// TIA Portal V19 program export: 9 tag tables, 2 data types, 63 data blocks, 26 code blocks (in call order from the OBs), 0 instance data blocks

VAR_GLOBAL   // PLC tag table "Default tag table"
   "System_Byte(1)" AT %MB1 : Byte;
   "Clock_Byte(1)" AT %MB0 : Byte;
   "Clock_10Hz(1)" AT %M0.0 : Bool;
   "Clock_5Hz(1)" AT %M0.1 : Bool;
   "Clock_2.5Hz(1)" AT %M0.2 : Bool;
   "Clock_2Hz(1)" AT %M0.3 : Bool;
   "Clock_1.25Hz(1)" AT %M0.4 : Bool;
   "Clock_1Hz(1)" AT %M0.5 : Bool;
   "Clock_0.625Hz(1)" AT %M0.6 : Bool;
   "Clock_0.5Hz(1)" AT %M0.7 : Bool;
END_VAR

VAR_GLOBAL   // PLC tag table "TT - Clocks"
   Clock_Byte AT %MB255 : Byte;
   Clock_10Hz AT %M255.0 : Bool;
   Clock_5Hz AT %M255.1 : Bool;
   "Clock_2.5Hz" AT %M255.2 : Bool;
   Clock_2Hz AT %M255.3 : Bool;
   "Clock_1.25Hz" AT %M255.4 : Bool;
   Clock_1Hz AT %M255.5 : Bool;
   "Clock_0.625Hz" AT %M255.6 : Bool;
   "Clock_0.5Hz" AT %M255.7 : Bool;
END_VAR

VAR_GLOBAL   // PLC tag table "TT - System"
   System_Byte AT %MB254 : Byte;
   FirstScan AT %M254.0 : Bool;
   DiagStatusUpdate AT %M254.1 : Bool;
   AlwaysTRUE AT %M254.2 : Bool;
   AlwaysFALSE AT %M254.3 : Bool;
END_VAR

VAR_GLOBAL   // PLC tag table "TT - Feeding"
   iFeedingSenCilOut_k1 AT %I2.4 : Bool;
   iFeedingSenLoaded AT %I2.5 : Bool;
   "oFeedingVenCilOut_K+" AT %Q1.5 : Bool;
END_VAR

VAR_GLOBAL   // PLC tag table "TT - General"
   iDkStart_S2 AT %I0.0 : Bool;   // NO
   iDkStop_S3 AT %I0.1 : Bool;   // NC
   iSelSchMan_Q2 AT %I0.2 : Bool;
   iDkReset_S4 AT %I0.3 : Bool;   // NO (reset VR)
   iStsNoodstop_S1 AT %I2.7 : Bool;   // NO
   oLmpAlarm_H1 AT %Q0.0 : Bool;
   oLmpWarningLowMaterial_H2 AT %Q1.7 : Bool;
   iSenPressure AT %I2.6 : Bool;   // true when pressure
END_VAR

VAR_GLOBAL   // PLC tag table "TT - Loading"
   iLoadingSenDown_a1 AT %I0.4 : Bool;
   iLoadingSenUp_a0 AT %I0.5 : Bool;
   iLoadingSenAtPick_b0 AT %I0.6 : Bool;
   iLoadingSenAtPlace_b1 AT %I0.7 : Bool;
   "oLoadingVenCilDown_A+" AT %Q0.1 : Bool;
   oLoadingVenCilPlace_B AT %Q0.2 : Bool;
   oLoadingVenGrip_C AT %Q0.3 : Bool;
END_VAR

VAR_GLOBAL   // PLC tag table "TT - Plate"
   iPlateSenCilPushingIn_d0 AT %I1.0 : Bool;   // Terugkoppeling pusher roteren plaat
   iPlateSenInductive_dm AT %I1.6 : Bool;   // True when metallic
   iPlateSenPresence_dp AT %I1.7 : Bool;
   iPlateSenNotBlack AT %I2.0 : Bool;   // Niet definitief, True when nothing and white
   "oPlateVenCilPushing_D+" AT %Q0.4 : Bool;
   "oPlateVenCilLocking_E+" AT %Q0.5 : Bool;
   "oPlateVenCilMeasuringDown_L+" AT %Q1.6 : Bool;
   iPlateSenHeight AT %IW65 : Int;
END_VAR

VAR_GLOBAL   // PLC tag table "TT - Reject"
   iRejectSenCilIn_f0 AT %I1.1 : Bool;
   iRejectSenCilOut_f1 AT %I1.2 : Bool;
   iRejectSenCilUp_g0 AT %I1.3 : Bool;
   "oRejectVenCilOut_F+" AT %Q0.6 : Bool;   // Bistabiel
   "oRejectVenCilIn_F-" AT %Q0.7 : Bool;   // Bistabiel
   oRejectVenCilDown_E AT %Q1.0 : Bool;
   "oRejectVenVacuum_V+" AT %Q1.1 : Bool;
   "iRejectSenVacuum_V+" AT %I2.1 : Bool;   // true when vacuum
END_VAR

VAR_GLOBAL   // PLC tag table "TT - Transport"
   iTransportSenDown_h1 AT %I1.4 : Bool;
   iTransportSenUp_h0 AT %I1.5 : Bool;
   iTransportSenAtPlate_i0 AT %I2.2 : Bool;
   iTransportSenAtCart_i1 AT %I2.3 : Bool;
   "oTransportVenCilDown_A+" AT %Q1.2 : Bool;
   "oTransportVenCilCart_I+" AT %Q1.3 : Bool;
   "oTransportVenGripClosed_J+" AT %Q1.4 : Bool;
END_VAR

TYPE "UDT_Recipe"
VERSION : 0.1
   STRUCT
      "Type" : Int;
      Aantal : Int;
      Progress : Int;
   END_STRUCT;

END_TYPE

TYPE "UDT_coverProperties"
VERSION : 0.1
   STRUCT
      loaded : Bool;   // Indicates that there is an item in the current location
      reject : Bool;   // Indicates that the current item is to be rejected
      properties : Struct
         metallic : Bool;   // Indicates that the current item is metallic
         notBlack : Bool;   // Indicates that the current item is not black
         correctOrientation : Bool;   // Indicates that the current item has the correct orientation
      END_STRUCT;
   END_STRUCT;

END_TYPE

DATA_BLOCK "DB_Alarm"
{ S7_Optimized_Access := 'TRUE' }
VERSION : 0.1
NON_RETAIN
   VAR 
      com : Struct   // Alarms from Transfer PLC communication
         S7_PUTerr : Bool;   // Error reported by PUT instruction
         S7_GETerr : Bool;   // Error reported by GET instruction
         WD : Bool;   // Watchdog timed out
      END_STRUCT;
      general : Struct   // General alarms
         global : Bool;   // Indicates that an alarm is active
         emergencyStop : Bool;   // Indicates that the emergency stop button is activated
         airPressure : Bool;   // Indicates a loss in air pressure
      END_STRUCT;
      feeding : Struct   // Alarms generated by the "Feeding" EM
         materialLow : Bool;   // Indicates an empty mag
      END_STRUCT;
      reject : Struct   // Alarms generated by the "Reject" EM
         vacuum : Bool;   // Indicates loss of vacuum when not expected
      END_STRUCT;
   END_VAR


BEGIN

END_DATA_BLOCK

DATA_BLOCK "DB_Global"
{ S7_Optimized_Access := 'TRUE' }
VERSION : 0.1
NON_RETAIN
   VAR 
      com : Struct   // Communication state object
         WD : Int;   // Watchdog mem for S7 communication with Transfer PLC
      END_STRUCT;
      general : Struct   // General state object
         startup : Bool;   // Indicates "startup" mode
         started : Bool;   // Indicates "started" mode
         man : Bool;   // Indicates "manual" mode
         resetSignal : Bool;   // Gives the reset signal (1s high)
         init : Bool;   // Sets the "Global Grafcet" to step 0
         DEBUG_AlwaysFalse : Bool;   // Used for debugging
         DEBUG_AlwaysTrue : Bool;   // Used for debugging
      END_STRUCT;
      feeding : Struct   // Feeding state object
         init : Bool;   // Sets the "Feeding Grafcet" to step 0
         sigReadyToReload : Bool;   // Indicates that "Feeding Grafcet" is ready
      END_STRUCT;
      loading : Struct   // Loading state object
         init : Bool;   // Sets the "Loading Grafcet" to step 0
         cmdPlaceNewCover : Bool;   // Command to start the "Loading" process
         sigReadyToPlace : Bool;   // Indicates that "Loading Grafcet" is ready
      END_STRUCT;
      plate : Struct   // Loading state object
         currentCovers { S7_SetPoint := 'False'} : Array[0..7] of "UDT_coverProperties";   // Array with all the data for the locations on the plate
         init_rotate : Bool;   // Sets the "Rotate Grafcet" to step 0
         cmdRotate : Bool;   // Command to start the "Rotate" process
         sigReadyToRotate : Bool;   // Indicates that "Rotate Grafcet" is ready
         init_measure : Bool;   // Sets the "Measure Grafcet" to step 0
         cmdMeasure : Bool;   // Command to start the "Measure" process
         sigReadyToMeasure : Bool;   // Indicates that "Measure Grafcet" is ready
      END_STRUCT;
      reject : Struct   // Reject state object
         init : Bool;   // Sets the "Reject Grafcet" to step 0
         cmdReject : Bool;   // Command to start the "Reject" process
         sigReadyToReject : Bool;   // Indicates that "Reject Grafcet" is ready
      END_STRUCT;
      transport : Struct   // Transport state object
         init : Bool;   // Sets the "Transport Grafcet" to step 0
         cmdTransport : Bool;   // Command to start the "Transport" process
         sigReadyToTransport : Bool;   // Indicates that "Transport Grafcet" is ready
      END_STRUCT;
   END_VAR


BEGIN

END_DATA_BLOCK

DATA_BLOCK "DB_IO"
{ S7_Optimized_Access := 'TRUE' }
VERSION : 0.1
NON_RETAIN
   VAR 
      general : Struct   // IO dedicated to no specific EM
         iDkStart : Bool;   // Processed input value
         iDkStop : Bool;   // Processed input value
         iSelSchMan : Bool;   // Processed input value
         iDkReset : Bool;   // Processed input value
         iSenPressure : Bool;   // Processed input value
         iStsNoodstop : Bool;   // Processed input value
         oLmpAlarm : Bool;   // Automatic output value
         oLmpWarningLowMaterial : Bool;   // Automatic output value
      END_STRUCT;
      feeding : Struct   // IO dedicated to Feeding EM
         iFeedingSenCilOut_k1 : Bool;   // Processed input value
         iFeedingSenLoaded : Bool;   // Processed input value
         "oFeedingVenCilOut_K+" : Bool;   // Automatic output value
      END_STRUCT;
      loading : Struct   // IO dedicated to Loading EM
         iLoadingSenDown : Bool;   // Processed input value
         iLoadingSenUp : Bool;   // Processed input value
         iLoadingSenAtPick : Bool;   // Processed input value
         iLoadingSenAtPlace : Bool;   // Processed input value
         oLoadingVenCilDown : Bool;   // Automatic output value
         oLoadingVenCilPlace : Bool;   // Automatic output value
         oLoadingVenGrip : Bool;   // Automatic output value
      END_STRUCT;
      plate : Struct   // IO dedicated to Plate EM
         iPlateSenCilPushingIn : Bool;   // Processed input value
         iPlateSenInductive : Bool;   // Processed input value
         iPlateSenPresence : Bool;   // Processed input value
         iPlateSenNotBlack : Bool;   // Processed input value
         iPlateSenHeight : Int;   // Processed input value
         oPlateVenCilPushing : Bool;   // Automatic output value
         oPlateVenCilLocking : Bool;   // Automatic output value
         oPlateVenCilMeasuringDown : Bool;   // Automatic output value
      END_STRUCT;
      reject : Struct   // IO dedicated to Reject EM
         iRejectSenCilIn : Bool;   // Processed input value
         iRejectSenCilOut : Bool;   // Processed input value
         iRejectSenCilUp : Bool;   // Processed input value
         iRejectSenVacuum : Bool;   // Processed input value
         oRejectVenCilOut : Bool;   // Automatic output value
         oRejectVenCilIn : Bool;   // Automatic output value
         oRejectVenCilDown : Bool;   // Automatic output value
         oRejectVenVacuum : Bool;   // Automatic output value
      END_STRUCT;
      transport : Struct   // IO dedicated to Transport EM
         iTransportSenDown : Bool;   // Processed input value
         iTransportSenUp : Bool;   // Processed input value
         iTransportSenAtPlate : Bool;   // Processed input value
         iTransportSenAtCart : Bool;   // Processed input value
         oTransportVenCilDown : Bool;   // Automatic output value
         oTransportVenCilCart : Bool;   // Automatic output value
         oTransportVenGripClosed : Bool;   // Automatic output value
      END_STRUCT;
   END_VAR


BEGIN

END_DATA_BLOCK

DATA_BLOCK "DB_Testing"
{ S7_Optimized_Access := 'TRUE' }
VERSION : 0.1
NON_RETAIN
   VAR 
      enable : Struct
         TransferPLC : Bool;   // Enables or disables the entire FB for testing purposes only
         GlobalGrafcet : Bool;   // Enables or disables the entire FB for testing purposes only
         Feeding : Bool;   // Enables or disables the entire FB for testing purposes only
         Loading : Bool;   // Enables or disables the entire FB for testing purposes only
         Rotate : Bool;   // Enables or disables the entire FB for testing purposes only
         Measure : Bool;   // Enables or disables the entire FB for testing purposes only
         Reject : Bool;   // Enables or disables the entire FB for testing purposes only
         Transport : Bool;   // Enables or disables the entire FB for testing purposes only
      END_STRUCT;
      init : Struct
         GlobalGrafcet : Bool;   // Sets current step to 0 (rising edge)
         Feeding : Bool;   // Sets current step to 0 (rising edge)
         Loading : Bool;   // Sets current step to 0 (rising edge)
         Rotate : Bool;   // Sets current step to 0 (rising edge)
         Measure : Bool;   // Sets current step to 0 (rising edge)
         Reject : Bool;   // Sets current step to 0 (rising edge)
         Transport : Bool;   // Sets current step to 0 (rising edge)
      END_STRUCT;
      value : Struct
         RecipeType : Int;   // Emulates current recipe to be 1 or 2 for testing purposes only
         RejectBit : Bool;   // Emulates that the current cover needs to be rejected
         CoverLoaded : Bool;   // Emulates that the location is loaded
      END_STRUCT;
      signal : Struct
         Transfer_CarrierReady : Bool;   // Emulates "carrierReady" signal from transfer PLC for testing purposes only
         Feeding_ReadyToReload : Bool;
         Loading_ReadyToPlace : Bool;
         Plate_ReadyToRotate : Bool;
         Plate_ReadyToMeasure : Bool;
         Reject_ReadyToReject : Bool;
         Transport_ReadyToTransport : Bool;
      END_STRUCT;
      cmd : Struct
         Loading : Bool;
         Plate_Rotate : Bool;
         Plate_Measure : Bool;
         Reject : Bool;
         Transport : Bool;
      END_STRUCT;
   END_VAR


BEGIN
   enable.TransferPLC := false;
   enable.GlobalGrafcet := false;
   enable.Feeding := false;
   enable.Loading := false;
   enable.Rotate := false;
   enable.Measure := false;
   enable.Reject := false;
   enable.Transport := false;
   init.GlobalGrafcet := false;
   init.Feeding := false;
   init.Loading := false;
   init.Rotate := false;
   init.Measure := false;
   init.Reject := false;
   init.Transport := false;
   value.RecipeType := 0;
   value.RejectBit := false;
   value.CoverLoaded := false;
   signal.Transfer_CarrierReady := false;
   signal.Feeding_ReadyToReload := false;
   signal.Loading_ReadyToPlace := false;
   signal.Plate_ReadyToRotate := false;
   signal.Plate_ReadyToMeasure := false;
   signal.Reject_ReadyToReject := false;
   signal.Transport_ReadyToTransport := false;
   cmd.Loading := false;
   cmd.Plate_Rotate := false;
   cmd.Plate_Measure := false;
   cmd.Reject := false;
   cmd.Transport := false;

END_DATA_BLOCK

DATA_BLOCK "DB_MES"
{ S7_Optimized_Access := 'FALSE' }
VERSION : 0.1
NON_RETAIN
   STRUCT 
      "IO van FB_ControlRecipes" : Struct
         iNewRecipe : Bool;
         iNewType : Int;
         iNewAantal : Int;
         iRemoveRecipe : Bool;
         iRecipeToBeRemoved : Int;
         iReceptKlaar : Bool;
         oFull : Bool;
         oEmpty : Bool;
      END_STRUCT;
      Algemeen : Struct
         mReceptGestart : Bool;
         mReceptActief : Bool;
         mInstallatieGestart : Bool;
         mWatchdogPLC : Int;
         mAlmActive : Bool;
      END_STRUCT;
      Alarmen : Struct
         mAlmGlobal : Bool;
         mAlmEmergencyStop : Bool;
         mAlmAirPressureLow : Bool;
         mAlmMaterialLow : Bool;
         mAlmVacuum : Bool;
      END_STRUCT;
      Merkers : Struct
         mMerkerSR1 : Bool;
         mMerkerSR2 : Bool;
      END_STRUCT;
   END_STRUCT;


BEGIN

END_DATA_BLOCK

DATA_BLOCK "DB_Recipes"
{ S7_Optimized_Access := 'FALSE' }
VERSION : 0.1
NON_RETAIN
   STRUCT 
      Recipes { S7_SetPoint := 'False'} : Array[0..4] of "UDT_Recipe";
   END_STRUCT;


BEGIN

END_DATA_BLOCK

DATA_BLOCK "FB_ControlRecipes_DB"
{ S7_Optimized_Access := 'TRUE' }
VERSION : 0.1
NON_RETAIN
"FB_ControlRecipes"

BEGIN

END_DATA_BLOCK

DATA_BLOCK "DB_HMI"
{ S7_Optimized_Access := 'TRUE' }
VERSION : 0.1
NON_RETAIN
   VAR 
      general : Struct
         read_fromPLC : Struct
            Gestart : Bool;
            Gestopt : Bool;
            Storing : Bool;
            Man : Bool;
            Auto : Bool;
         END_STRUCT;
         alarmen : Struct
            Emergency : Bool;
            AirPressure : Bool;
         END_STRUCT;
         write_toPLC : Struct
            Cmd_Start : Bool;   // Om te sturen in Auto
            Cmd_Stop : Bool;   // Om te sturen in Auto
            Cmd_Reset : Bool;   // Om te sturen in Auto
            Cmd_Init : Bool;
         END_STRUCT;
      END_STRUCT;
      feeding : Struct
         read_fromPLC : Struct
            SenLoaded : Bool;
            SenCilOut_k1 : Bool;
            MagazijnLeeg : Bool;
         END_STRUCT;
         alarmen : Struct
            MaterialLow : Bool;
         END_STRUCT;
         write_toPLC : Struct
            Man_Out : Bool;
         END_STRUCT;
      END_STRUCT;
      loading : Struct
         read_fromPLC : Struct
            SenDown_a1 : Bool;
            SenUp_a0 : Bool;
            SenAtPick_b0 : Bool;
            SenAtPlace_b1 : Bool;
            oGrip : Bool;   // Inlezen om weer te geven wat deze doet
         END_STRUCT;
         alarmen : Struct
            CilDownTimeout : Bool;
            CilPlaceTimeout : Bool;
         END_STRUCT;
         write_toPLC : Struct
            Man_Grip : Bool;
            Man_Down : Bool;
            Man_Place : Bool;
         END_STRUCT;
      END_STRUCT;
      plate : Struct
         read_fromPLC : Struct
            oLock : Bool;   // Inlezen om weer te geven wat deze doet
            SenCilPushIn : Bool;   // cylinder terug (not pushed) true
            oMeasureDown : Bool;   // cylinder uit Measure
            MeasureDownNOK : Bool;   // Berekend
            MeasureDownOK : Bool;   // Berekend
         END_STRUCT;
         alarmen : Struct
            CilMeasureTime : Bool;
         END_STRUCT;
         write_toPLC : Struct
            Man_Measure : Bool;
            Man_Push : Bool;
            Man_Lock : Bool;
         END_STRUCT;
      END_STRUCT;
      reject : Struct
         read_fromPLC : Struct
            SenVacuüm : Bool;
            SenOut : Bool;
            SenIn : Bool;
            SenUp : Bool;
         END_STRUCT;
         alarmen : Struct
            CilOutTime : Bool;
            Vacuüm : Bool;
         END_STRUCT;
         write_toPLC : Struct
            Man_Out : Bool;
            Man_Vacuüm : Bool;
            Man_Down : Bool;
         END_STRUCT;
      END_STRUCT;
      transport : Struct
         read_fromPLC : Struct
            oGrip : Bool;   // inlezen om weer te geven wat deze doet
            CilUp : Bool;
            CilDown : Bool;
            CilPick : Bool;
            CilPlace : Bool;
         END_STRUCT;
         alarmen : Struct
            CilDownTime : Bool;
            CilPlaceTime : Bool;
         END_STRUCT;
         write_toPLC : Struct
            Man_Grip : Bool;
            Man_Down : Bool;
            Man_Place : Bool;
         END_STRUCT;
      END_STRUCT;
   END_VAR


BEGIN

END_DATA_BLOCK

DATA_BLOCK "DB_TransferPLC"
{ S7_Optimized_Access := 'TRUE' }
VERSION : 0.1
NON_RETAIN
   VAR 
      Watchdog : Int;   // value between 0 and 20000 that counts up every second
      CarrierReady : Bool;   // inidcates if the carrier is in place and ready to recieve a cover
      ItemPlaced : Bool;   // indicates if the cover station has placed the cover on the carrier
   END_VAR


BEGIN

END_DATA_BLOCK

DATA_BLOCK "ID_PE_GlobalGrafcet"
{ S7_Optimized_Access := 'TRUE' }
VERSION : 0.1
NON_RETAIN
"FB_PE_GlobalGrafcet"

BEGIN

END_DATA_BLOCK

DATA_BLOCK "ID_PE_Feeding_Grafcet"
{ S7_Optimized_Access := 'TRUE' }
VERSION : 0.1
NON_RETAIN
"FB_PE_Feeding_Grafcet"

BEGIN

END_DATA_BLOCK

DATA_BLOCK "ID_PE_Loading_Grafcet"
{ S7_Optimized_Access := 'TRUE' }
VERSION : 0.1
NON_RETAIN
"FB_PE_Loading"

BEGIN

END_DATA_BLOCK

DATA_BLOCK "ID_PE_Plate_Grafcet"
{ S7_Optimized_Access := 'TRUE' }
VERSION : 0.1
NON_RETAIN
"FB_PE_Plate_Rotate"

BEGIN

END_DATA_BLOCK

DATA_BLOCK "ID_PE_Plate_Measure"
{ S7_Optimized_Access := 'TRUE' }
VERSION : 0.1
NON_RETAIN
"FB_PE_Plate_Measure"

BEGIN

END_DATA_BLOCK

DATA_BLOCK "ID_PE_Reject"
{ S7_Optimized_Access := 'TRUE' }
VERSION : 0.1
NON_RETAIN
"FB_PE_Reject"

BEGIN

END_DATA_BLOCK

DATA_BLOCK "ID_PE_Transport"
{ S7_Optimized_Access := 'TRUE' }
VERSION : 0.1
NON_RETAIN
"FB_PE_Transport"

BEGIN

END_DATA_BLOCK

DATA_BLOCK "ID_Algemeen_CM_DI_iDkReset"
{ S7_Optimized_Access := 'FALSE' }
VERSION : 0.1
NON_RETAIN
"FB_CM_DI_Sensor"

BEGIN

END_DATA_BLOCK

DATA_BLOCK "ID_Algemeen_CM_DI_iDkStart"
{ S7_Optimized_Access := 'FALSE' }
VERSION : 0.1
NON_RETAIN
"FB_CM_DI_Sensor"

BEGIN

END_DATA_BLOCK

DATA_BLOCK "ID_Algemeen_CM_DI_iDkStop"
{ S7_Optimized_Access := 'FALSE' }
VERSION : 0.1
NON_RETAIN
"FB_CM_DI_Sensor"

BEGIN

END_DATA_BLOCK

DATA_BLOCK "ID_Algemeen_CM_DI_iSelSchMan"
{ S7_Optimized_Access := 'FALSE' }
VERSION : 0.1
NON_RETAIN
"FB_CM_DI_Sensor"

BEGIN

END_DATA_BLOCK

DATA_BLOCK "ID_Algemeen_CM_DI_iStsNoodstop"
{ S7_Optimized_Access := 'FALSE' }
VERSION : 0.1
NON_RETAIN
"FB_CM_DI_Sensor"

BEGIN

END_DATA_BLOCK

DATA_BLOCK "ID_Algemeen_PE_StartStop"
{ S7_Optimized_Access := 'FALSE' }
VERSION : 0.1
NON_RETAIN
"FB_PE_StartStop"

BEGIN

END_DATA_BLOCK

DATA_BLOCK "ID_CM_Lamp_Alarm_H1"
{ S7_Optimized_Access := 'TRUE' }
VERSION : 0.1
NON_RETAIN
"FB_CM_Lamp_1200"

BEGIN

END_DATA_BLOCK

DATA_BLOCK "ID_Feeding_CM_DI_SenCilOut"
{ S7_Optimized_Access := 'FALSE' }
VERSION : 0.1
NON_RETAIN
"FB_CM_DI_Sensor"

BEGIN

END_DATA_BLOCK

DATA_BLOCK "ID_Feeding_CM_DI_SenLoaded"
{ S7_Optimized_Access := 'FALSE' }
VERSION : 0.1
NON_RETAIN
"FB_CM_DI_Sensor"

BEGIN

END_DATA_BLOCK

DATA_BLOCK "ID_Feeding_CM_oFeedingVenCilOut"
{ S7_Optimized_Access := 'FALSE' }
VERSION : 0.1
NON_RETAIN
"FB_CM_Cilinder"

BEGIN

END_DATA_BLOCK

DATA_BLOCK "ID_Loading_CM_DI_iLoadingSenAtPick_b0"
{ S7_Optimized_Access := 'FALSE' }
VERSION : 0.1
NON_RETAIN
"FB_CM_DI_Sensor"

BEGIN

END_DATA_BLOCK

DATA_BLOCK "ID_Loading_CM_DI_iLoadingSenAtPlace_b1"
{ S7_Optimized_Access := 'FALSE' }
VERSION : 0.1
NON_RETAIN
"FB_CM_DI_Sensor"

BEGIN

END_DATA_BLOCK

DATA_BLOCK "ID_Loading_CM_DI_iLoadingSenDown_a1"
{ S7_Optimized_Access := 'FALSE' }
VERSION : 0.1
NON_RETAIN
"FB_CM_DI_Sensor"

BEGIN

END_DATA_BLOCK

DATA_BLOCK "ID_Loading_CM_DI_iLoadingSenUp_a0"
{ S7_Optimized_Access := 'FALSE' }
VERSION : 0.1
NON_RETAIN
"FB_CM_DI_Sensor"

BEGIN

END_DATA_BLOCK

DATA_BLOCK "ID_Loading_CM_oLoadingVenCilDown_A+"
{ S7_Optimized_Access := 'FALSE' }
VERSION : 0.1
NON_RETAIN
"FB_CM_Cilinder"

BEGIN

END_DATA_BLOCK

DATA_BLOCK "ID_Loading_CM_oLoadingVenCilPlace_B"
{ S7_Optimized_Access := 'FALSE' }
VERSION : 0.1
NON_RETAIN
"FB_CM_Cilinder"

BEGIN

END_DATA_BLOCK

DATA_BLOCK "ID_Loading_CM_oLoadingVenGrip_C"
{ S7_Optimized_Access := 'FALSE' }
VERSION : 0.1
NON_RETAIN
"FB_CM_Cilinder"

BEGIN

END_DATA_BLOCK

DATA_BLOCK "ID_Plate_CM_DI_iPlateSenCilPushingIn_d0"
{ S7_Optimized_Access := 'FALSE' }
VERSION : 0.1
NON_RETAIN
"FB_CM_DI_Sensor"

BEGIN

END_DATA_BLOCK

DATA_BLOCK "ID_Plate_CM_DI_iPlateSenInductive_dm"
{ S7_Optimized_Access := 'FALSE' }
VERSION : 0.1
NON_RETAIN
"FB_CM_DI_Sensor"

BEGIN

END_DATA_BLOCK

DATA_BLOCK "ID_Plate_CM_DI_iPlateSenNotBlack"
{ S7_Optimized_Access := 'FALSE' }
VERSION : 0.1
NON_RETAIN
"FB_CM_DI_Sensor"

BEGIN

END_DATA_BLOCK

DATA_BLOCK "ID_Plate_CM_DI_iPlateSenPresence_dp"
{ S7_Optimized_Access := 'FALSE' }
VERSION : 0.1
NON_RETAIN
"FB_CM_DI_Sensor"

BEGIN

END_DATA_BLOCK

DATA_BLOCK "ID_Plate_CM_oPlateVenCilLocking_E+"
{ S7_Optimized_Access := 'FALSE' }
VERSION : 0.1
NON_RETAIN
"FB_CM_Cilinder"

BEGIN

END_DATA_BLOCK

DATA_BLOCK "ID_Plate_CM_oPlateVenCilMeasuringDown_L+"
{ S7_Optimized_Access := 'FALSE' }
VERSION : 0.1
NON_RETAIN
"FB_CM_Cilinder"

BEGIN

END_DATA_BLOCK

DATA_BLOCK "ID_Plate_CM_oPlateVenCilPushing_D+"
{ S7_Optimized_Access := 'FALSE' }
VERSION : 0.1
NON_RETAIN
"FB_CM_Cilinder"

BEGIN

END_DATA_BLOCK

DATA_BLOCK "ID_Reject_CM_DI_iRejectSenCilIn_f0"
{ S7_Optimized_Access := 'FALSE' }
VERSION : 0.1
NON_RETAIN
"FB_CM_DI_Sensor"

BEGIN

END_DATA_BLOCK

DATA_BLOCK "ID_Reject_CM_DI_iRejectSenCilOut_f1"
{ S7_Optimized_Access := 'FALSE' }
VERSION : 0.1
NON_RETAIN
"FB_CM_DI_Sensor"

BEGIN

END_DATA_BLOCK

DATA_BLOCK "ID_Reject_CM_DI_iRejectSenCilUp_g0"
{ S7_Optimized_Access := 'FALSE' }
VERSION : 0.1
NON_RETAIN
"FB_CM_DI_Sensor"

BEGIN

END_DATA_BLOCK

DATA_BLOCK "ID_Reject_CM_DI_iRejectSenVacuum_V+"
{ S7_Optimized_Access := 'FALSE' }
VERSION : 0.1
NON_RETAIN
"FB_CM_DI_Sensor"

BEGIN

END_DATA_BLOCK

DATA_BLOCK "ID_Reject_CM_oRejectVenCilDown_E"
{ S7_Optimized_Access := 'FALSE' }
VERSION : 0.1
NON_RETAIN
"FB_CM_Cilinder"

BEGIN

END_DATA_BLOCK

DATA_BLOCK "ID_Reject_CM_oRejectVenCilOutIn"
{ S7_Optimized_Access := 'FALSE' }
VERSION : 0.1
NON_RETAIN
"FB_CM_Cilinder"

BEGIN

END_DATA_BLOCK

DATA_BLOCK "ID_Reject_CM_oRejectVenVacuum_V+"
{ S7_Optimized_Access := 'FALSE' }
VERSION : 0.1
NON_RETAIN
"FB_CM_Cilinder"

BEGIN

END_DATA_BLOCK

DATA_BLOCK "ID_Transport_CM_DI_iTransportSenAtCart_i1"
{ S7_Optimized_Access := 'FALSE' }
VERSION : 0.1
NON_RETAIN
"FB_CM_DI_Sensor"

BEGIN

END_DATA_BLOCK

DATA_BLOCK "ID_Transport_CM_DI_iTransportSenAtPlate_i0"
{ S7_Optimized_Access := 'FALSE' }
VERSION : 0.1
NON_RETAIN
"FB_CM_DI_Sensor"

BEGIN

END_DATA_BLOCK

DATA_BLOCK "ID_Transport_CM_DI_iTransportSenDown_h1"
{ S7_Optimized_Access := 'FALSE' }
VERSION : 0.1
NON_RETAIN
"FB_CM_DI_Sensor"

BEGIN

END_DATA_BLOCK

DATA_BLOCK "ID_Transport_CM_DI_iTransportSenUp_h0"
{ S7_Optimized_Access := 'FALSE' }
VERSION : 0.1
NON_RETAIN
"FB_CM_DI_Sensor"

BEGIN

END_DATA_BLOCK

DATA_BLOCK "ID_Transport_CM_oTransportVenCilCart_I+"
{ S7_Optimized_Access := 'FALSE' }
VERSION : 0.1
NON_RETAIN
"FB_CM_Cilinder"

BEGIN

END_DATA_BLOCK

DATA_BLOCK "ID_Transport_CM_oTransportVenCilDown_A+"
{ S7_Optimized_Access := 'FALSE' }
VERSION : 0.1
NON_RETAIN
"FB_CM_Cilinder"

BEGIN

END_DATA_BLOCK

DATA_BLOCK "ID_Transport_CM_oTransportVenGripClosed_J+"
{ S7_Optimized_Access := 'FALSE' }
VERSION : 0.1
NON_RETAIN
"FB_CM_Cilinder"

BEGIN

END_DATA_BLOCK

DATA_BLOCK "ID_GET_fromTransferPLC"
{InstructionName := 'GET';
 LibVersion := '1.3';
 S7_Optimized_Access := 'TRUE' }
AUTHOR : SIMATIC
FAMILY : COM_FUNC
NAME : GET
VERSION : 1.1
NON_RETAIN
GET

BEGIN

END_DATA_BLOCK

DATA_BLOCK "ID_PUT_toTransferPLC"
{InstructionName := 'PUT';
 LibVersion := '1.3';
 S7_Optimized_Access := 'TRUE' }
AUTHOR : SIMATIC
FAMILY : COM_FUNC
NAME : PUT
VERSION : 1.1
NON_RETAIN
PUT

BEGIN

END_DATA_BLOCK

DATA_BLOCK "ID_TON_ResetSignal"
{InstructionName := 'IEC_TIMER';
 LibVersion := '1.0';
 S7_Optimized_Access := 'TRUE' }
AUTHOR : Simatic
FAMILY : IEC
NAME : IEC_TMR
VERSION : 1.0
NON_RETAIN
IEC_TIMER

BEGIN

END_DATA_BLOCK

DATA_BLOCK "ID_TON_TransferPLCWatchdog"
{InstructionName := 'IEC_TIMER';
 LibVersion := '1.0';
 S7_Optimized_Access := 'TRUE' }
AUTHOR : Simatic
FAMILY : IEC
NAME : IEC_TMR
VERSION : 1.0
NON_RETAIN
IEC_TIMER

BEGIN

END_DATA_BLOCK

DATA_BLOCK "ID_TP_ResetSignal"
{InstructionName := 'IEC_TIMER';
 LibVersion := '1.0';
 S7_Optimized_Access := 'TRUE' }
AUTHOR : Simatic
FAMILY : IEC
NAME : IEC_TMR
VERSION : 1.0
NON_RETAIN
IEC_TIMER

BEGIN

END_DATA_BLOCK

DATA_BLOCK "IEC_Counter_0_DB"
{InstructionName := 'IEC_COUNTER';
 LibVersion := '1.0';
 S7_Optimized_Access := 'TRUE' }
AUTHOR : Simatic
FAMILY : IEC
NAME : CNTR
VERSION : 1.0
IEC_COUNTER

BEGIN

END_DATA_BLOCK

DATA_BLOCK "R_TRIG_DB"
{InstructionName := 'R_TRIG';
 LibVersion := '1.0';
 S7_Optimized_Access := 'TRUE' }
AUTHOR : SIMATIC
FAMILY : BIT
NAME : R_TRIG
VERSION : 1.0
NON_RETAIN
R_TRIG

BEGIN

END_DATA_BLOCK

DATA_BLOCK "R_TRIG_DB_1"
{InstructionName := 'R_TRIG';
 LibVersion := '1.0';
 S7_Optimized_Access := 'TRUE' }
AUTHOR : SIMATIC
FAMILY : BIT
NAME : R_TRIG
VERSION : 1.0
NON_RETAIN
R_TRIG

BEGIN

END_DATA_BLOCK

DATA_BLOCK "R_TRIG_DB_2"
{InstructionName := 'R_TRIG';
 LibVersion := '1.0';
 S7_Optimized_Access := 'TRUE' }
AUTHOR : SIMATIC
FAMILY : BIT
NAME : R_TRIG
VERSION : 1.0
NON_RETAIN
R_TRIG

BEGIN

END_DATA_BLOCK

ORGANIZATION_BLOCK "Main"   // OB1, FBD, ProgramCycle
TITLE = "Main Program Sweep (Cycle)"
{ S7_Optimized_Access := 'TRUE' }
// stored: SetENOAutomatically false
   VAR_INPUT
      Initial_Call : Bool;   // Initial call of this OB
      Remanence : Bool;   // =True, if remanent data are available
   END_VAR
   VAR_TEMP   // added for the SCL form of the ladder/FBD networks
      _w1 : Bool;
   END_VAR
BEGIN

REGION Network 1: Debug tags
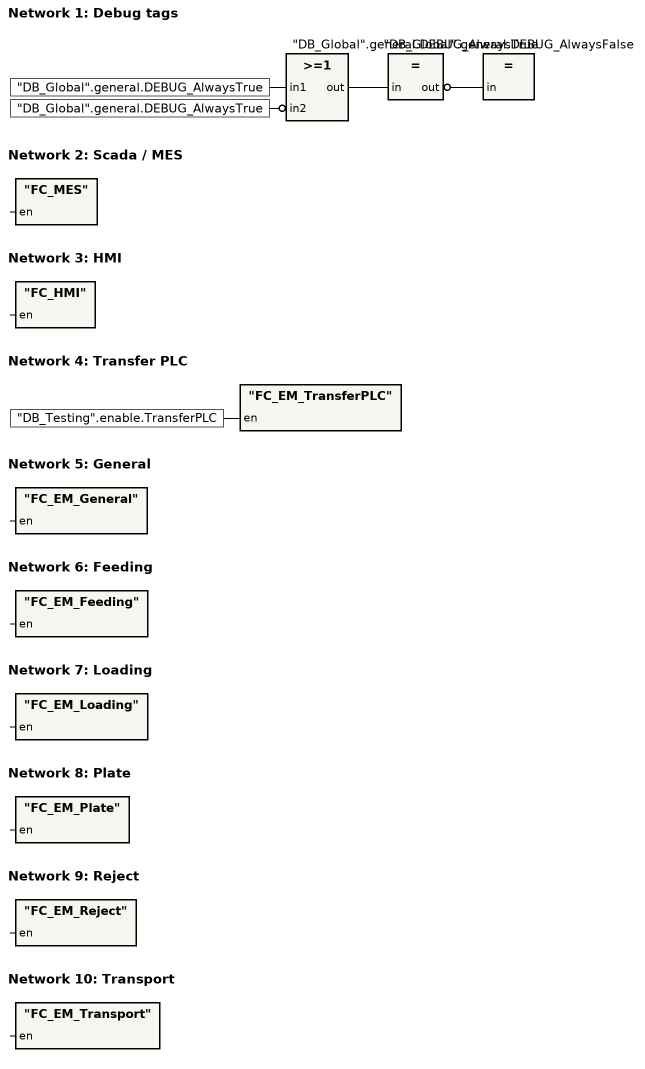
   #_w1 := "DB_Global".general.DEBUG_AlwaysTrue OR NOT "DB_Global".general.DEBUG_AlwaysTrue;
   "DB_Global".general.DEBUG_AlwaysTrue := #_w1;
   "DB_Global".general.DEBUG_AlwaysFalse := NOT #_w1;
END_REGION

REGION Network 2: Scada / MES
   "FC_MES"();
END_REGION

REGION Network 3: HMI
   "FC_HMI"();
END_REGION

REGION Network 4: Transfer PLC
   IF "DB_Testing".enable.TransferPLC THEN "FC_EM_TransferPLC"(); END_IF;
END_REGION

REGION Network 5: General
   "FC_EM_General"();
END_REGION

REGION Network 6: Feeding
   "FC_EM_Feeding"();
END_REGION

REGION Network 7: Loading
   "FC_EM_Loading"();
END_REGION

REGION Network 8: Plate
   "FC_EM_Plate"();
END_REGION

REGION Network 9: Reject
   "FC_EM_Reject"();
END_REGION

REGION Network 10: Transport
   "FC_EM_Transport"();
END_REGION
END_ORGANIZATION_BLOCK

FUNCTION "FC_MES" : Void   // FC8, FBD
{ S7_Optimized_Access := 'TRUE' }
// stored: SetENOAutomatically false
BEGIN

REGION Network 1: managen van recipes
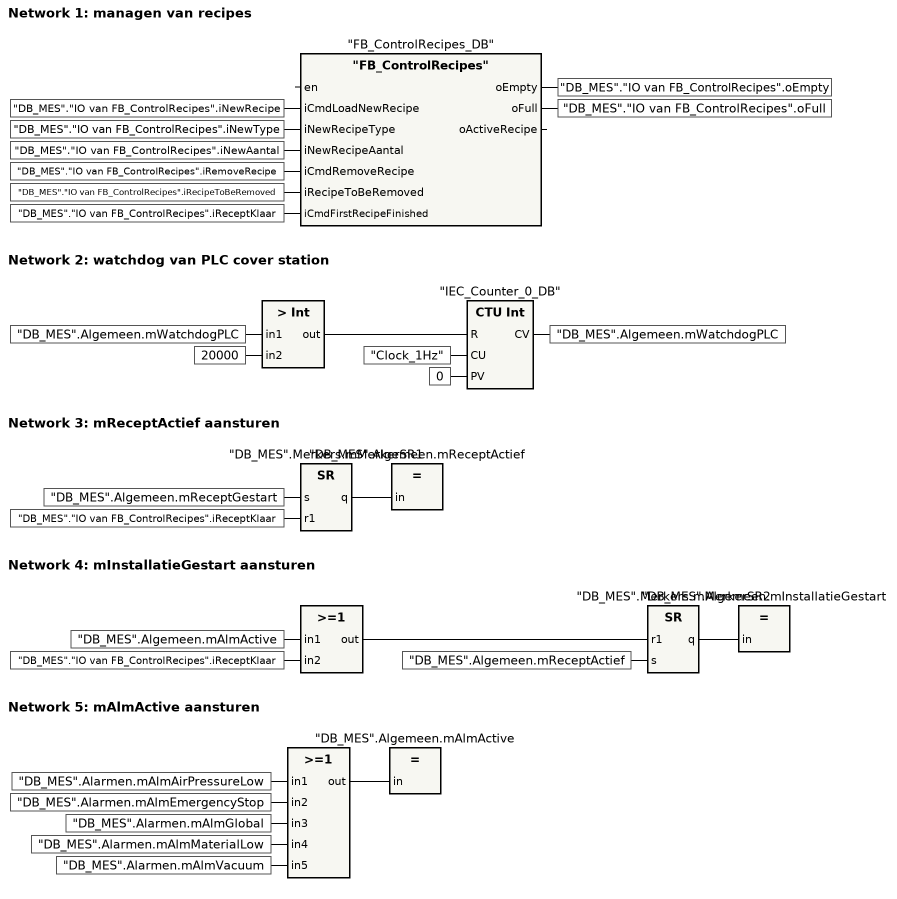
   "FB_ControlRecipes_DB"(iCmdLoadNewRecipe := "DB_MES"."IO van FB_ControlRecipes".iNewRecipe,   // "FB_ControlRecipes"
                          iNewRecipeType := "DB_MES"."IO van FB_ControlRecipes".iNewType,
                          iNewRecipeAantal := "DB_MES"."IO van FB_ControlRecipes".iNewAantal,
                          iCmdRemoveRecipe := "DB_MES"."IO van FB_ControlRecipes".iRemoveRecipe,
                          iRecipeToBeRemoved := "DB_MES"."IO van FB_ControlRecipes".iRecipeToBeRemoved,
                          iCmdFirstRecipeFinished := "DB_MES"."IO van FB_ControlRecipes".iReceptKlaar,
                          oEmpty => "DB_MES"."IO van FB_ControlRecipes".oEmpty,
                          oFull => "DB_MES"."IO van FB_ControlRecipes".oFull);
END_REGION

REGION Network 2: watchdog van PLC cover station
   "IEC_Counter_0_DB".CTU(R := "DB_MES".Algemeen.mWatchdogPLC > 20000,
                          CU := "Clock_1Hz",
                          PV := 0,
                          CV => "DB_MES".Algemeen.mWatchdogPLC);
END_REGION

REGION Network 3: mReceptActief aansturen
   IF "DB_MES".Algemeen.mReceptGestart THEN
       "DB_MES".Merkers.mMerkerSR1 := TRUE;   // SR flip-flop
   END_IF;
   IF "DB_MES"."IO van FB_ControlRecipes".iReceptKlaar THEN "DB_MES".Merkers.mMerkerSR1 := FALSE; END_IF;
   "DB_MES".Algemeen.mReceptActief := "DB_MES".Merkers.mMerkerSR1;
END_REGION

REGION Network 4: mInstallatieGestart aansturen
   IF "DB_MES".Algemeen.mReceptActief THEN
       "DB_MES".Merkers.mMerkerSR2 := TRUE;   // SR flip-flop
   END_IF;
   IF "DB_MES".Algemeen.mAlmActive OR "DB_MES"."IO van FB_ControlRecipes".iReceptKlaar THEN
       "DB_MES".Merkers.mMerkerSR2 := FALSE;
   END_IF;
   "DB_MES".Algemeen.mInstallatieGestart := "DB_MES".Merkers.mMerkerSR2;
END_REGION

REGION Network 5: mAlmActive aansturen
   "DB_MES".Algemeen.mAlmActive := "DB_MES".Alarmen.mAlmAirPressureLow OR "DB_MES".Alarmen.mAlmEmergencyStop OR "DB_MES".Alarmen.mAlmGlobal OR "DB_MES".Alarmen.mAlmMaterialLow OR "DB_MES".Alarmen.mAlmVacuum;
END_REGION

REGION Network 6: schrijven naar node-red
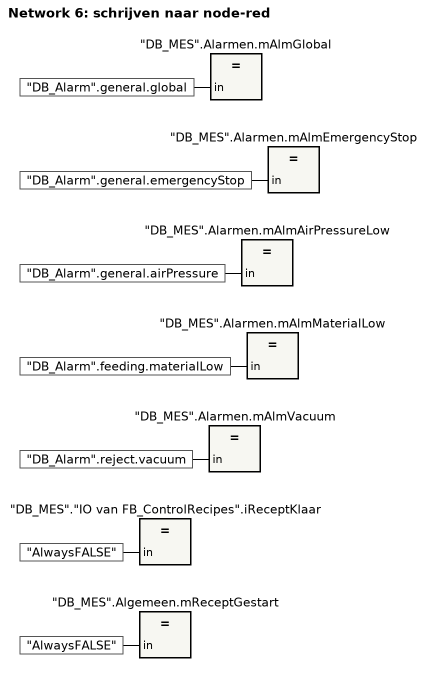
   "DB_MES".Alarmen.mAlmGlobal := "DB_Alarm".general.global;
   "DB_MES".Alarmen.mAlmEmergencyStop := "DB_Alarm".general.emergencyStop;
   "DB_MES".Alarmen.mAlmAirPressureLow := "DB_Alarm".general.airPressure;
   "DB_MES".Alarmen.mAlmMaterialLow := "DB_Alarm".feeding.materialLow;
   "DB_MES".Alarmen.mAlmVacuum := "DB_Alarm".reject.vacuum;
   "DB_MES"."IO van FB_ControlRecipes".iReceptKlaar := "AlwaysFALSE";
   "DB_MES".Algemeen.mReceptGestart := "AlwaysFALSE";
END_REGION
END_FUNCTION

FUNCTION_BLOCK "FB_ControlRecipes"
{ S7_Optimized_Access := 'TRUE' }
VERSION : 0.1
   VAR_INPUT 
      iCmdLoadNewRecipe : Bool;
      iNewRecipeType : Int;   // 1 of 2 (zwart/metaal)
      iNewRecipeAantal : Int;
      iCmdRemoveRecipe : Bool;
      iRecipeToBeRemoved : Int;   // 0, 1, 2, 3 of 4
      iCmdFirstRecipeFinished : Bool;   // wordt door PLC zelf hoog gezet
   END_VAR

   VAR_OUTPUT 
      oEmpty : Bool;
      oFull : Bool;
      oActiveRecipe : "UDT_Recipe";
   END_VAR

   VAR 
      sFreeSlots : Int;
      i1 : Int;
      i2 : Int;
      i3 : Int;
      sAddRecipe : Bool;
      sRemoveRecipe : Bool;
      sFirstRecipeFinished : Bool;
   END_VAR


BEGIN
	REGION General
	    
	    //positive trigger om nieuw recept toe te voegen
	    "R_TRIG_DB"(CLK := #iCmdLoadNewRecipe,
	                Q => #sAddRecipe);
	    
	    //positive trigger om recept te verwijderen
	    "R_TRIG_DB_1"(CLK:=#iCmdRemoveRecipe,
	                  Q=>#sRemoveRecipe);
	    
	    //positive trigger als eerste recept klaar is
	    "R_TRIG_DB_2"(CLK:=#iCmdFirstRecipeFinished,
	                  Q=>#sFirstRecipeFinished);
	    
	    //aantal lege slots bepalen in DB_Recipes adhv #i1
	    #sFreeSlots := 0;
	    FOR #i1 := 0 TO 4 DO
	        IF "DB_Recipes".Recipes[#i1].Type = 0 THEN
	            #sFreeSlots := #sFreeSlots + 1;
	        END_IF;
	    END_FOR;
	    
	    //full hoog zetten als er 5 recepten in wachtrij staan
	    IF #sFreeSlots = 0 THEN
	        #oFull := 1;
	    ELSE
	        #oFull := 0;
	    END_IF;
	    
	    //empty hoog zetten als er geen recepten in de wachtrij staan
	    IF #sFreeSlots = 5 THEN
	        #oEmpty := 1;
	    ELSE
	        #oEmpty := 0;
	    END_IF;
	    
	    //schrijven naar oActiveRecipe
	    #oActiveRecipe.Type := "DB_Recipes".Recipes[0].Type;
	    #oActiveRecipe.Aantal := "DB_Recipes".Recipes[0].Aantal;
	    
	END_REGION
	
	REGION Add
	    
	    //schrijven naar DB_Recipes als er plaats is
	    IF NOT(#sFreeSlots = 0) THEN
	        //toevoegen van nieuw recept en resetten van inputs type/aantal
	        IF #sAddRecipe THEN
	            "DB_Recipes".Recipes[5 - #sFreeSlots].Type := #iNewRecipeType;
	            "DB_Recipes".Recipes[5 - #sFreeSlots].Aantal := #iNewRecipeAantal;
	            "DB_MES"."IO van FB_ControlRecipes".iNewType := 0;
	            "DB_MES"."IO van FB_ControlRecipes".iNewAantal := 0;
	        END_IF;
	    END_IF;
	 
	END_REGION
	
	REGION Remove
	    
	    //een recept verwijderen
	    IF #sRemoveRecipe THEN
	        //alle recepten een plaats opschuiven
	        FOR #i2 := (#iRecipeToBeRemoved -1) TO 3 DO
	            "DB_Recipes".Recipes[#i2] := "DB_Recipes".Recipes[#i2 + 1];
	        END_FOR;
	        //allerlaatste recept leegmaken en #iRecipeToBeRemoved resetten
	        "DB_Recipes".Recipes[4].Type := 0;
	        "DB_Recipes".Recipes[4].Aantal := 0;
	        "DB_Recipes".Recipes[4].Progress := 0;
	        "DB_MES"."IO van FB_ControlRecipes".iRecipeToBeRemoved := 0;
	    END_IF;
	    
	    //het eerste recept verwijderen als deze uitgevoerd is
	    IF #sFirstRecipeFinished THEN
	        "DB_Recipes".Recipes[0] := "DB_Recipes".Recipes[1];
	        "DB_Recipes".Recipes[1] := "DB_Recipes".Recipes[2];
	        "DB_Recipes".Recipes[2] := "DB_Recipes".Recipes[3];
	        "DB_Recipes".Recipes[3] := "DB_Recipes".Recipes[4];
	        "DB_Recipes".Recipes[4].Type := 0;
	        "DB_Recipes".Recipes[4].Aantal := 0;
	        "DB_Recipes".Recipes[4].Progress := 0;
	    END_IF;
	   
	END_REGION
END_FUNCTION_BLOCK

FUNCTION "FC_HMI" : Void
{ S7_Optimized_Access := 'TRUE' }
VERSION : 0.1
   VAR CONSTANT 
      TODO : Bool := false;
   END_VAR


BEGIN
	REGION General
	    
	    REGION Read from PLC
	        "DB_HMI".general.read_fromPLC.Gestart := "DB_Global".general.started;
	        "DB_HMI".general.read_fromPLC.Gestopt := NOT "DB_Global".general.started; // Nodig?
	        "DB_HMI".general.read_fromPLC.Storing := "DB_Alarm".general.global;
	        "DB_HMI".general.read_fromPLC.Auto := NOT "DB_Global".general.man;
	    END_REGION
	    
	    REGION Alarmen
	        "DB_HMI".general.alarmen.Emergency := "DB_Alarm".general.global; // Dubbel
	        "DB_HMI".general.alarmen.AirPressure := "DB_Alarm".general.airPressure;
	    END_REGION
	    
	    REGION Write to PLC
	        // Zie FC_EM_General "DB_HMI".general.write_toPLC.Cmd_Start
	        // Zie FC_EM_General "DB_HMI".general.write_toPLC.Cmd_Stop
	        // Zie FC_EM_General "DB_HMI".general.write_toPLC.Cmd_Reset
	    END_REGION
	    
	END_REGION
	
	REGION Feeding
	    
	    REGION Read from PLC
	        "DB_HMI".feeding.read_fromPLC.SenLoaded := "DB_IO".feeding.iFeedingSenLoaded;
	        "DB_HMI".feeding.read_fromPLC.SenCilOut_k1 := "DB_IO".feeding.iFeedingSenCilOut_k1;
	        "DB_HMI".feeding.read_fromPLC.MagazijnLeeg := "DB_Alarm".feeding.materialLow;
	    END_REGION
	    
	    REGION Alarmen
	        
	       
	        "DB_HMI".feeding.alarmen.MaterialLow := "DB_Alarm".feeding.materialLow; 
	    END_REGION
	    
	    REGION Write to PLC
	        // Zie FC_EM_Feeding "DB_HMI".feeding.write_toPLC.Man_Out
	    END_REGION
	    
	END_REGION
	
	REGION Loading
	    
	    REGION Read from PLC
	        "DB_HMI".loading.read_fromPLC.SenDown_a1 := "DB_IO".loading.iLoadingSenDown;
	        "DB_HMI".loading.read_fromPLC.SenUp_a0 := "DB_IO".loading.iLoadingSenUp;
	        "DB_HMI".loading.read_fromPLC.SenAtPick_b0 := "DB_IO".loading.iLoadingSenAtPick;
	        "DB_HMI".loading.read_fromPLC.SenAtPlace_b1 := "DB_IO".loading.iLoadingSenAtPlace;
	        "DB_HMI".loading.read_fromPLC.oGrip := "oLoadingVenGrip_C";
	    END_REGION
	    
	    REGION Alarmen
	        "DB_HMI".loading.alarmen.CilDownTimeout := #TODO;
	        
	        "DB_HMI".loading.alarmen.CilPlaceTimeout := #TODO;
	        
	    END_REGION
	    
	    REGION Write to PLC
	        // Zie FC_EM_Loading "DB_HMI".loading.write_toPLC.Man_Grip
	        // Zie FC_EM_Loading "DB_HMI".loading.write_toPLC.Man_Down
	        // Zie FC_EM_Loading "DB_HMI".loading.write_toPLC.Man_Place
	    END_REGION
	    
	END_REGION
	
	REGION Plate
	    
	    REGION Read from PLC
	        "DB_HMI".plate.read_fromPLC.oLock := "oPlateVenCilLocking_E+";
	        "DB_HMI".plate.read_fromPLC.SenCilPushIn := "DB_IO".plate.iPlateSenCilPushingIn;
	        "DB_HMI".plate.read_fromPLC.oMeasureDown := "oPlateVenCilMeasuringDown_L+";
	        
	    END_REGION
	    
	    REGION Alarmen
	        
	        "DB_HMI".plate.alarmen.CilMeasureTime := #TODO;
	       
	    END_REGION
	    
	    REGION Write to PLC
	        // Zie FC_EM_Plate "DB_HMI".plate.write_toPLC.Man_Measure
	        // Zie FC_EM_Plate "DB_HMI".plate.write_toPLC.Man_Push
	        // Zie FC_EM_Plate "DB_HMI".plate.write_toPLC.Man_Lock
	    END_REGION
	    
	END_REGION
	
	REGION Reject
	    
	    REGION Read from PLC
	        "DB_HMI".reject.read_fromPLC.SenVacuüm := "DB_IO".reject.iRejectSenVacuum;
	        "DB_HMI".reject.read_fromPLC.SenOut := "DB_IO".reject.iRejectSenCilOut;
	        "DB_HMI".reject.read_fromPLC.SenIn := "DB_IO".reject.iRejectSenCilIn;
	        "DB_HMI".reject.read_fromPLC.SenUp := "DB_IO".reject.iRejectSenCilUp;
	    END_REGION
	    
	    REGION Alarmen
	        "DB_HMI".reject.alarmen.CilOutTime := #TODO;
	       
	        
	        "DB_HMI".reject.alarmen.Vacuüm := "DB_Alarm".reject.vacuum; // Valid IMO
	    END_REGION
	    
	    REGION Write to PLC
	        // Zie FC_EM_Reject "DB_HMI".reject.write_toPLC.Man_Out
	        // Zie FC_EM_Reject "DB_HMI".reject.write_toPLC.Man_Vacuüm
	        // Zie FC_EM_Reject "DB_HMI".reject.write_toPLC.Man_Down
	    END_REGION
	    
	END_REGION
	
	REGION Transport
	    
	    REGION Read from PLC
	        "DB_HMI".transport.read_fromPLC.oGrip := "oTransportVenGripClosed_J+";
	        "DB_HMI".transport.read_fromPLC.CilUp := "DB_IO".transport.iTransportSenUp;
	        "DB_HMI".transport.read_fromPLC.CilDown := "DB_IO".transport.iTransportSenDown;
	        "DB_HMI".transport.read_fromPLC.CilPick := "DB_IO".transport.iTransportSenAtPlate;
	        "DB_HMI".transport.read_fromPLC.CilPlace := "DB_IO".transport.iTransportSenAtCart;
	    END_REGION
	    
	    REGION Alarmen
	        "DB_HMI".transport.alarmen.CilDownTime := #TODO;
	        
	        "DB_HMI".transport.alarmen.CilPlaceTime := #TODO;
	       
	    END_REGION
	    
	    REGION Write to PLC
	        // Zie FC_EM_Transport "DB_HMI".transport.write_toPLC.Man_Grip
	        // Zie FC_EM_Transport "DB_HMI".transport.write_toPLC.Man_Down
	        // Zie FC_EM_Transport "DB_HMI".transport.write_toPLC.Man_Place
	    END_REGION
	    
	END_REGION
END_FUNCTION

FUNCTION "FC_EM_TransferPLC" : Void
{ S7_Optimized_Access := 'TRUE' }
VERSION : 0.1

BEGIN
	REGION Get
	    "ID_GET_fromTransferPLC"(ID := W#16#100, // S7 connection ID
	                             REQ := "Clock_1Hz", // Read on Rising Edge
	                             
	                             // Pointer to "readyToRecieve" bit in Transfer PLC
	                             ADDR_1 := P#DB66.DBX0.0 Bool 1,
	                             RD_1 := "DB_TransferPLC".CarrierReady,
	                             
	                             // Pointer to "watchdog" int in Transfer PLC
	                             ADDR_2 := P#DB66.DBX2.0 Int 1,
	                             RD_2 := "DB_TransferPLC".Watchdog,
	                             
	                             ERROR => "DB_Alarm".com.S7_GETerr);
	END_REGION
	
	REGION Put
	    "ID_PUT_toTransferPLC"(ID := W#16#100, // S7 connection ID
	                           REQ := "Clock_1Hz", // Read on Rising Edge
	                           
	                           // Pointer to "itemPlaced" bit in Transfer PLC
	                           ADDR_1 := P#DB66.DBX0.0 Bool 1,
	                           SD_1 := "DB_TransferPLC".ItemPlaced,
	                           
	                           ERROR => "DB_Alarm".com.S7_PUTerr);
	END_REGION
	                        
	REGION Watchdog
	    "ID_TON_TransferPLCWatchdog".TON(IN := "DB_TransferPLC".Watchdog = "DB_Global".com.WD,
	                                     PT := T#2s,
	                                     Q => "DB_Alarm".com.WD);
	    
	    "DB_Global".com.WD := "DB_TransferPLC".Watchdog;
	END_REGION
END_FUNCTION

FUNCTION "FC_EM_General" : Void   // FC1, FBD
TITLE = FC Algemeen
{ S7_Optimized_Access := 'TRUE' }
// stored: SetENOAutomatically false
   VAR_TEMP
      xFlashPeriod : Real;
   END_VAR
BEGIN

REGION Network 1: ------------------------------------------------------------------------ Inputs ------------------------------------------------------------------------
END_REGION

REGION Network 2: Verwerken van iStsNoodstop
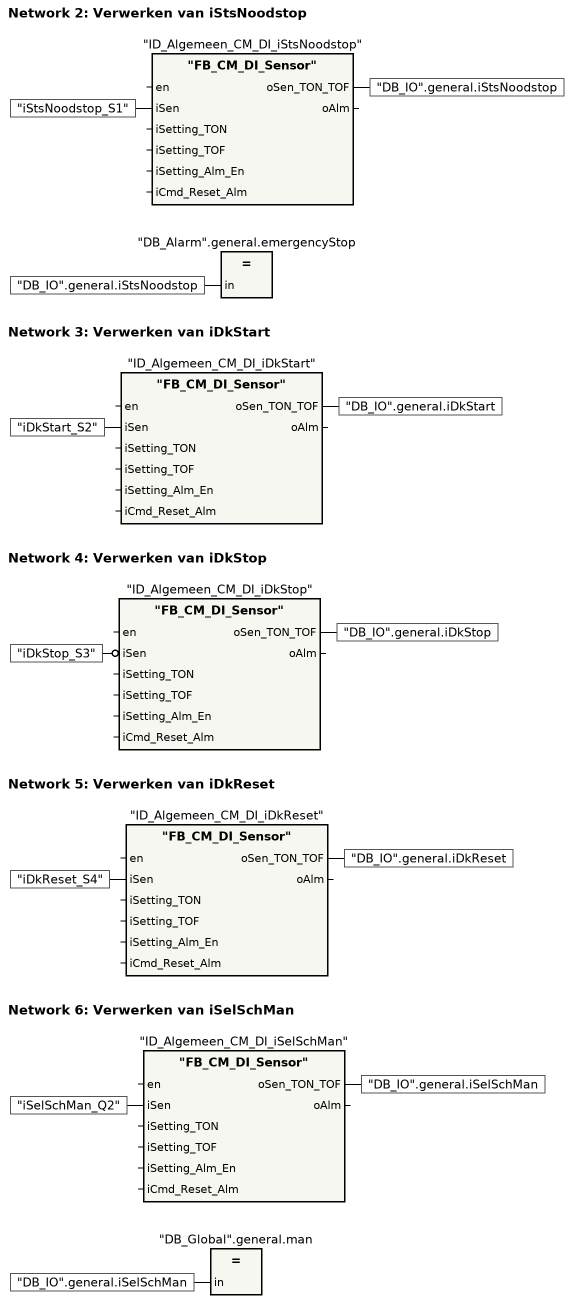
   "ID_Algemeen_CM_DI_iStsNoodstop"(iSen := "iStsNoodstop_S1", oSen_TON_TOF => "DB_IO".general.iStsNoodstop);   // "FB_CM_DI_Sensor"
   "DB_Alarm".general.emergencyStop := "DB_IO".general.iStsNoodstop;
END_REGION

REGION Network 3: Verwerken van iDkStart
   "ID_Algemeen_CM_DI_iDkStart"(iSen := "iDkStart_S2", oSen_TON_TOF => "DB_IO".general.iDkStart);   // "FB_CM_DI_Sensor"
END_REGION

REGION Network 4: Verwerken van iDkStop
   "ID_Algemeen_CM_DI_iDkStop"(iSen := NOT "iDkStop_S3", oSen_TON_TOF => "DB_IO".general.iDkStop);   // "FB_CM_DI_Sensor"
END_REGION

REGION Network 5: Verwerken van iDkReset
   "ID_Algemeen_CM_DI_iDkReset"(iSen := "iDkReset_S4", oSen_TON_TOF => "DB_IO".general.iDkReset);   // "FB_CM_DI_Sensor"
END_REGION

REGION Network 6: Verwerken van iSelSchMan
   "ID_Algemeen_CM_DI_iSelSchMan"(iSen := "iSelSchMan_Q2", oSen_TON_TOF => "DB_IO".general.iSelSchMan);   // "FB_CM_DI_Sensor"
   "DB_Global".general.man := "DB_IO".general.iSelSchMan;
END_REGION

REGION Network 7: ------------------------------------------------------------------------ Logic -------------------------------------------------------------------------
END_REGION

REGION Network 8: Start/stop logica van de installatie
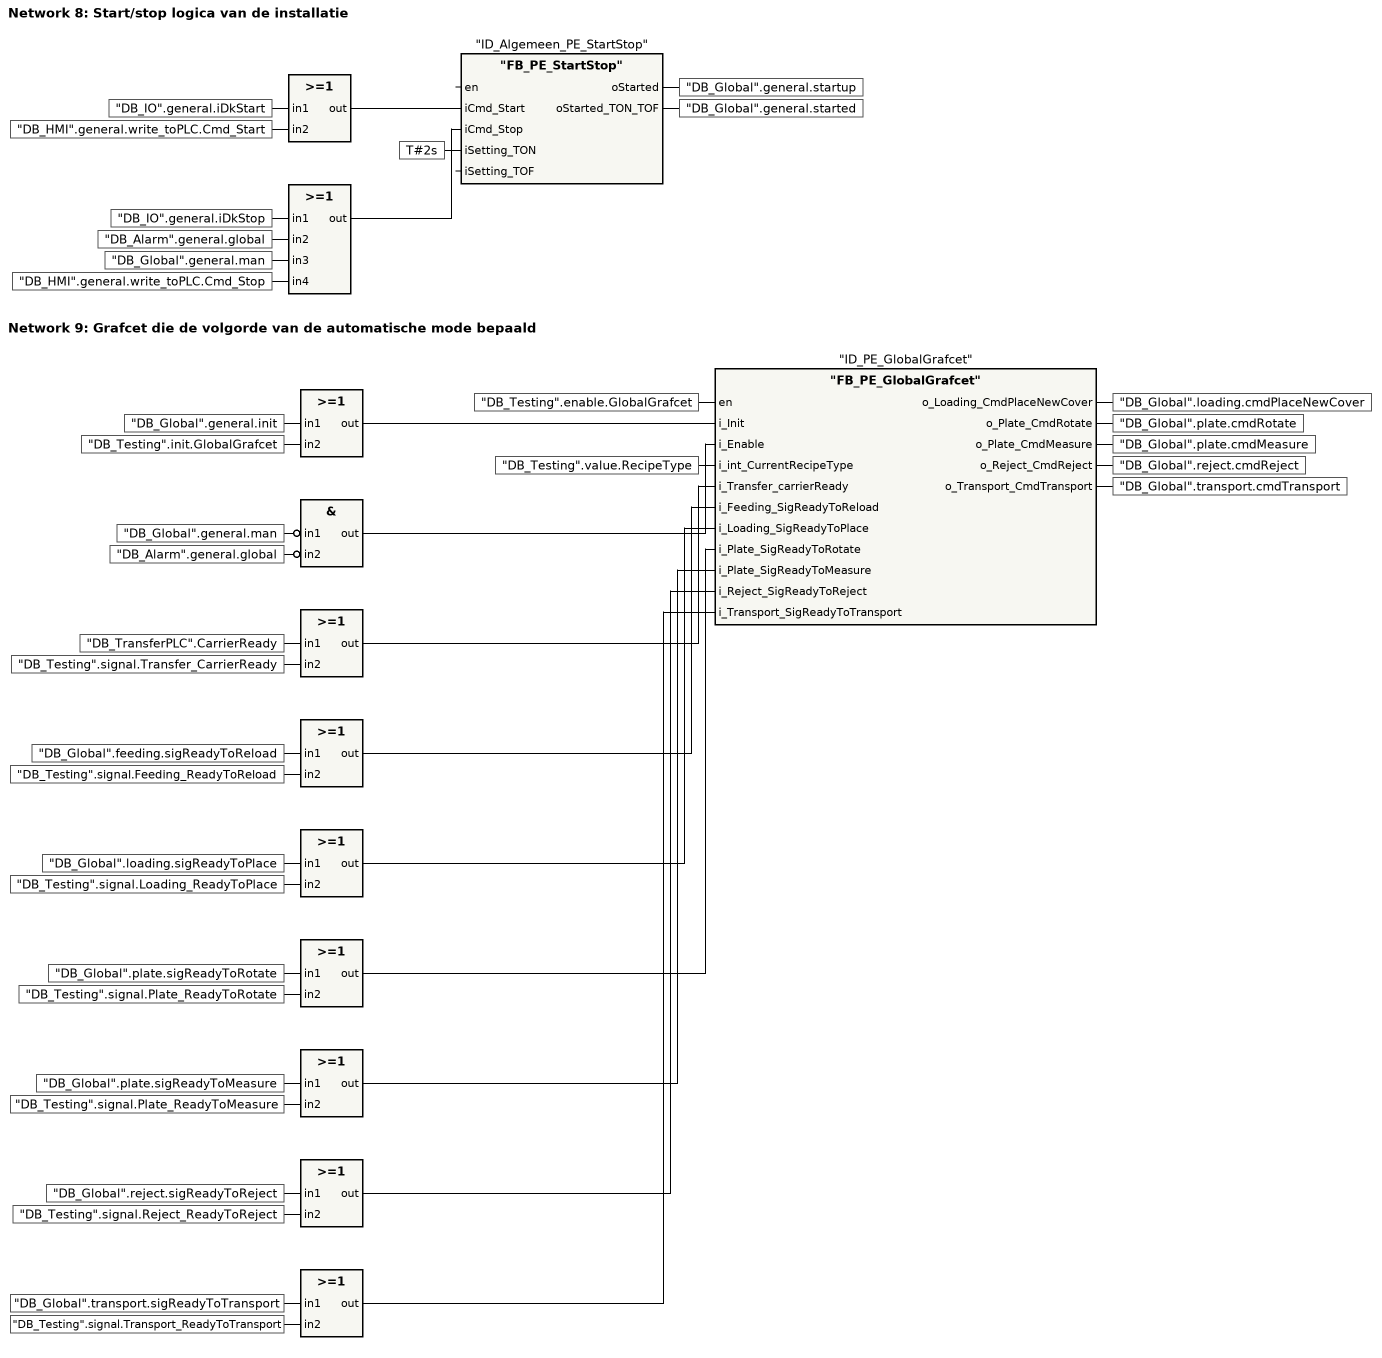
   "ID_Algemeen_PE_StartStop"(iCmd_Start := "DB_IO".general.iDkStart OR "DB_HMI".general.write_toPLC.Cmd_Start,   // "FB_PE_StartStop"
                           iCmd_Stop := "DB_IO".general.iDkStop OR "DB_Alarm".general.global OR "DB_Global".general.man OR "DB_HMI".general.write_toPLC.Cmd_Stop,
                           iSetting_TON := T#2s,
                           oStarted => "DB_Global".general.startup,
                           oStarted_TON_TOF => "DB_Global".general.started);
END_REGION

REGION Network 9: Grafcet die de volgorde van de automatische mode bepaald
   IF "DB_Testing".enable.GlobalGrafcet THEN
       "ID_PE_GlobalGrafcet"(i_Init := "DB_Global".general.init OR "DB_Testing".init.GlobalGrafcet,   // "FB_PE_GlobalGrafcet"
                             i_Enable := NOT "DB_Global".general.man AND NOT "DB_Alarm".general.global,
                             i_int_CurrentRecipeType := "DB_Testing".value.RecipeType,
                             i_Transfer_carrierReady := "DB_TransferPLC".CarrierReady OR "DB_Testing".signal.Transfer_CarrierReady,
                             i_Feeding_SigReadyToReload := "DB_Global".feeding.sigReadyToReload OR "DB_Testing".signal.Feeding_ReadyToReload,
                             i_Loading_SigReadyToPlace := "DB_Global".loading.sigReadyToPlace OR "DB_Testing".signal.Loading_ReadyToPlace,
                             i_Plate_SigReadyToRotate := "DB_Global".plate.sigReadyToRotate OR "DB_Testing".signal.Plate_ReadyToRotate,
                             i_Plate_SigReadyToMeasure := "DB_Global".plate.sigReadyToMeasure OR "DB_Testing".signal.Plate_ReadyToMeasure,
                             i_Reject_SigReadyToReject := "DB_Global".reject.sigReadyToReject OR "DB_Testing".signal.Reject_ReadyToReject,
                             i_Transport_SigReadyToTransport := "DB_Global".transport.sigReadyToTransport OR "DB_Testing".signal.Transport_ReadyToTransport,
                             o_Loading_CmdPlaceNewCover => "DB_Global".loading.cmdPlaceNewCover,
                             o_Plate_CmdRotate => "DB_Global".plate.cmdRotate,
                             o_Plate_CmdMeasure => "DB_Global".plate.cmdMeasure,
                             o_Reject_CmdReject => "DB_Global".reject.cmdReject,
                             o_Transport_CmdTransport => "DB_Global".transport.cmdTransport);
   END_IF;
END_REGION

REGION Network 10: ----------------------------------------------------------------------- Signals -----------------------------------------------------------------------
END_REGION

REGION Network 11: Genereren van reset puls
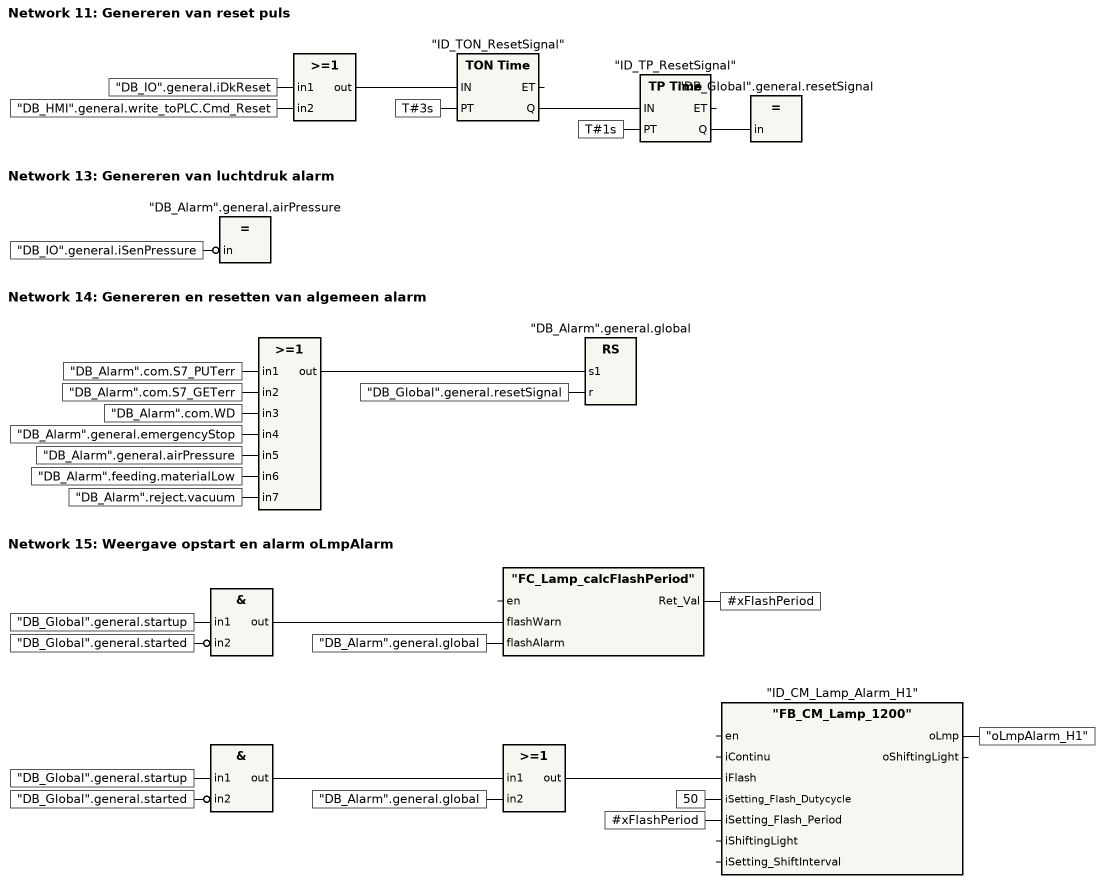
   "ID_TON_ResetSignal".TON(IN := "DB_IO".general.iDkReset OR "DB_HMI".general.write_toPLC.Cmd_Reset,
                           PT := T#3s);
   "ID_TP_ResetSignal".TP(IN := "ID_TON_ResetSignal".Q, PT := T#1s);
   "DB_Global".general.resetSignal := "ID_TP_ResetSignal".Q;
END_REGION

REGION Network 12: --------------------------------------------------------------------- Alarms ------------------------------------------------------------------------
END_REGION

REGION Network 13: Genereren van luchtdruk alarm
   "DB_Alarm".general.airPressure := NOT "DB_IO".general.iSenPressure;
END_REGION

REGION Network 14: Genereren en resetten van algemeen alarm
   IF "DB_Global".general.resetSignal THEN
       "DB_Alarm".general.global := FALSE;   // RS flip-flop
   END_IF;
   IF "DB_Alarm".com.S7_PUTerr OR "DB_Alarm".com.S7_GETerr OR "DB_Alarm".com.WD OR "DB_Alarm".general.emergencyStop OR "DB_Alarm".general.airPressure OR "DB_Alarm".feeding.materialLow OR "DB_Alarm".reject.vacuum THEN
       "DB_Alarm".general.global := TRUE;
   END_IF;
END_REGION

REGION Network 15: Weergave opstart en alarm oLmpAlarm
   #xFlashPeriod := "FC_Lamp_calcFlashPeriod"(flashWarn := "DB_Global".general.startup AND NOT "DB_Global".general.started,
                           flashAlarm := "DB_Alarm".general.global);
   "ID_CM_Lamp_Alarm_H1"(iFlash := ("DB_Global".general.startup AND NOT "DB_Global".general.started) OR "DB_Alarm".general.global,   // "FB_CM_Lamp_1200"
                         iSetting_Flash_Dutycycle := 50,
                         iSetting_Flash_Period := #xFlashPeriod,
                         oLmp => "oLmpAlarm_H1");
END_REGION
END_FUNCTION

FUNCTION_BLOCK "FB_CM_DI_Sensor"
{ S7_Optimized_Access := 'FALSE' }
VERSION : 0.1
   VAR_INPUT 
      iSen { S7_HiddenAssignment := 'Show'} : Bool;   // Sensor input signal
      iSetting_TON : Time;   // On-delay time for oSen_TO
      iSetting_TOF : Time;   // Off-delay time for oSen_TO
      iSetting_Alm_En { S7_HiddenAssignment := 'Hide'} : Bool;   // Activate alarm functionality
      iCmd_Reset_Alm { S7_HiddenAssignment := 'Hide'} : Bool;   // Command to reset the alarm
   END_VAR

   VAR_OUTPUT 
      oSen_TON_TOF : Bool;   // Sensor with delays signal
      oAlm { S7_HiddenAssignment := 'Hide'} : Bool;   // Alarm sensor actived
   END_VAR

   VAR 
      sAlm : Bool;   // Alarm sensor actived retain > compliant Machine Directive 2006/42/EG
      sTON_Sen {InstructionName := 'TON_TIME'; LibVersion := '1.0'} : TON_TIME;
      sTOF_Sen {InstructionName := 'TOF_TIME'; LibVersion := '1.0'} : TOF_TIME;
   END_VAR


BEGIN
	REGION Sensor 
	    //Optional delays on sensor
	    #sTON_Sen(IN := #iSen,
	          PT := #iSetting_TON);
	    #sTOF_Sen(IN:=#sTON_Sen.Q,
	          PT:=#iSetting_TOF);
	    //Output result
	    #oSen_TON_TOF:= #sTOF_Sen.Q;
	END_REGION
	
	REGION Alarm  
	    //Sensor alarm circuit
	    IF #iCmd_Reset_Alm THEN
	        #sAlm := FALSE;
	    END_IF;
	    //Cause after reset = Priority on cause > compliant Machine Directive 2006/42/EG
	    IF #iSetting_Alm_En AND #sTON_Sen.Q THEN
	        #sAlm := TRUE;
	    END_IF;
	    //Output result
	    #oAlm := #sAlm;
	END_REGION ;
END_FUNCTION_BLOCK

FUNCTION_BLOCK "FB_PE_StartStop"   // FB30, FBD
TITLE = Start-stop procedure
{ S7_Optimized_Access := 'FALSE' }
// stored: AutoNumber false, SetENOAutomatically false
   VAR_INPUT
      iCmd_Start : Bool;   // Start command
      iCmd_Stop : Bool;   // Stop command
      iSetting_TON : Time;   // On-delay time for oStarted_TO
      iSetting_TOF : Time;   // Off-delay time for oStarted_TO
   END_VAR
   VAR_OUTPUT
      oStarted : Bool;   // Started signal
      oStarted_TON_TOF : Bool;   // Started with delays signal
   END_VAR
   VAR
      sRE_CmdStart { S7_SetPoint := 'True'} : Bool;
      sStarted { S7_SetPoint := 'True'} : Bool;   // Started not-retain > Automatic restart not allowed during power failures > compliant Machine Directive 2006/42/EG
      sTON_Started { S7_SetPoint := 'True'} : TON_TIME;
      sTOF_Started { S7_SetPoint := 'True'} : TOF_TIME;
   END_VAR
   VAR_TEMP   // added for the SCL form of the ladder/FBD networks
      _w1 : Bool;
   END_VAR
BEGIN

REGION Network 1: Start-stop circuit
   // (**Rising edge on iCmdStart > compliant Machine Directive 2006/42/EG
   // 1) To prevent a reasonably foreseenable human error that could lead to a dangerous situation
   //    Human error = To brigde the start button
   // 2) To prevent that errors in the control logic leads to a dangerous situation
   //    Error in the control logic = Short circuit in the start circuit**)
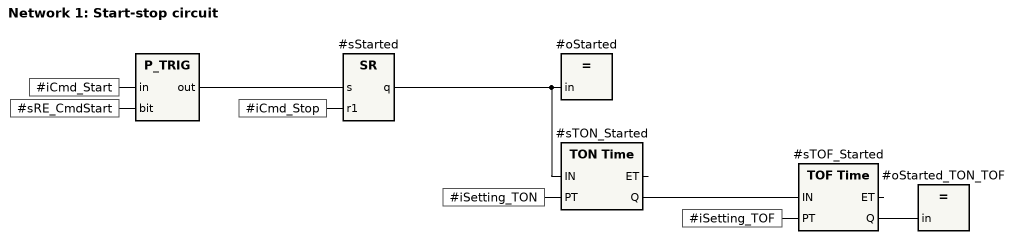
   #_w1 := #iCmd_Start AND NOT #sRE_CmdStart;   // rising edge
   #sRE_CmdStart := #iCmd_Start;
   IF #_w1 THEN
       #sStarted := TRUE;   // SR flip-flop
   END_IF;
   IF #iCmd_Stop THEN #sStarted := FALSE; END_IF;
   #oStarted := #sStarted;
   #sTON_Started(IN := #sStarted, PT := #iSetting_TON);   // TON
   #sTOF_Started(IN := #sTON_Started.Q, PT := #iSetting_TOF);   // TOF
   #oStarted_TON_TOF := #sTOF_Started.Q;
END_REGION
END_FUNCTION_BLOCK

FUNCTION_BLOCK "FB_PE_GlobalGrafcet"
{ S7_Optimized_Access := 'TRUE' }
VERSION : 0.1
   VAR_INPUT 
      i_Init : Bool;
      i_Enable : Bool;
      i_int_CurrentRecipeType : Int;
      i_Transfer_carrierReady : Bool;
      i_Feeding_SigReadyToReload : Bool;
      i_Loading_SigReadyToPlace : Bool;
      i_Plate_SigReadyToRotate : Bool;
      i_Plate_SigReadyToMeasure : Bool;
      i_Reject_SigReadyToReject : Bool;
      i_Transport_SigReadyToTransport : Bool;
   END_VAR

   VAR_OUTPUT 
      o_Loading_CmdPlaceNewCover : Bool;
      o_Plate_CmdRotate : Bool;
      o_Plate_CmdMeasure : Bool;
      o_Reject_CmdReject : Bool;
      o_Transport_CmdTransport : Bool;
   END_VAR

   VAR 
      sStep : Int;
      sInit : Bool;
      sEdge_2to3 : Bool;
   END_VAR

   VAR_TEMP 
      xEdge_2to3 : Bool;
   END_VAR


BEGIN
	REGION init
	    IF #i_Init AND NOT(#sInit = #i_Init) THEN
	        #sStep := 0;
	    END_IF;
	    #sInit := #i_Init;
	END_REGION
	
	REGION enable
	    IF NOT #i_Enable THEN
	        GOTO afterGrafcetLogic;
	    END_IF;
	END_REGION
	
	REGION edge detection
	    
	    REGION 2 to 3
	        // Always false
	        #xEdge_2to3 := FALSE;
	        // Edge detect
	        IF
	            #i_Plate_SigReadyToRotate
	            AND NOT #sEdge_2to3
	        THEN
	            #xEdge_2to3 := TRUE;
	        END_IF;
	        // Set equal for next check
	        #sEdge_2to3 := #i_Plate_SigReadyToRotate;
	    END_REGION
	    
	END_REGION
	
	REGION grafcet logic
	    CASE #sStep OF
	        0:
	            IF
	                ( #i_int_CurrentRecipeType = 1 OR #i_int_CurrentRecipeType = 2)
	                AND #i_Feeding_SigReadyToReload
	                AND #i_Loading_SigReadyToPlace
	                AND #i_Plate_SigReadyToRotate
	                AND #i_Plate_SigReadyToMeasure
	                AND #i_Reject_SigReadyToReject
	                AND #i_Transport_SigReadyToTransport
	            THEN
	                #sStep := 1;
	            END_IF;
	        1:
	            #sStep := 2;
	        2:
	            IF #xEdge_2to3 THEN
	                #sStep := 3;
	            END_IF;
	        3:
	            #sStep := 4;
	        4:
	            IF
	                #i_Reject_SigReadyToReject
	                AND #i_Transfer_carrierReady
	            THEN
	                #sStep := 5;
	            END_IF;
	        5:
	            #sStep := 6;
	        6:
	            IF
	                #i_Transport_SigReadyToTransport
	                AND #i_Loading_SigReadyToPlace
	                AND #i_Plate_SigReadyToMeasure
	            THEN
	                #sStep := 0;
	            END_IF;
	        ELSE
	            #sStep := 0;
	    END_CASE;
	    
	END_REGION
	
	afterGrafcetLogic: // Jump destination
	
	REGION outputs
	    
	    #o_Loading_CmdPlaceNewCover := #sStep = 3;
	    #o_Plate_CmdRotate := #sStep = 1;
	    #o_Plate_CmdMeasure := #sStep = 3;
	    #o_Reject_CmdReject := #sStep = 3;
	    #o_Transport_CmdTransport := #sStep = 5;
	                   
	END_REGION
	
END_FUNCTION_BLOCK

FUNCTION "FC_Lamp_calcFlashPeriod" : Real
{ S7_Optimized_Access := 'TRUE' }
VERSION : 0.1
   VAR_INPUT 
      flashWarn : Bool;
      flashAlarm : Bool;
   END_VAR

   VAR_TEMP 
      xPeriod : Real;
   END_VAR


BEGIN
	IF #flashAlarm THEN
	    #xPeriod := 0.5;
	ELSIF #flashWarn THEN
	    #xPeriod := 1.0;
	ELSE
	    #xPeriod := 2.0;
	END_IF;
	
	#FC_Lamp_calcFlashPeriod := #xPeriod;
END_FUNCTION

FUNCTION_BLOCK "FB_CM_Lamp_1200"
{ S7_Optimized_Access := 'TRUE' }
VERSION : 0.1
   VAR_INPUT 
      iContinu : Bool;
      iFlash : Bool;
      iSetting_Flash_Dutycycle : USInt;   // Duty cycle in %
      iSetting_Flash_Period : Real;   // Periode in seconden
      iShiftingLight { S7_HiddenAssignment := 'Hide'} : Bool;   // Looplicht
      iSetting_ShiftInterval { S7_HiddenAssignment := 'Hide'} : Real;   // Tijd tussen de opschuivende bits
   END_VAR

   VAR_OUTPUT 
      oLmp : Bool;
      oShiftingLight { S7_HiddenAssignment := 'Hide'} : Byte;
   END_VAR

   VAR 
      R_Trig_StartFlash {InstructionName := 'R_TRIG'; LibVersion := '1.0'} : R_TRIG;
      Timer_Flash_LmpOff {InstructionName := 'TP_TIME'; LibVersion := '1.0'} : TP_TIME;
      F_TRIG_Flash_LmpOff {InstructionName := 'F_TRIG'; LibVersion := '1.0'} : F_TRIG;
      Timer_Flash_LmpOn {InstructionName := 'TP_TIME'; LibVersion := '1.0'} : TP_TIME;
      F_TRIG_Flash_LmpOn {InstructionName := 'F_TRIG'; LibVersion := '1.0'} : F_TRIG;
      F_Edge_FlashLmpOff { S7_SetPoint := 'True'} : Bool;
      R_Edge_StartFlash : Bool;
      F_Edge_FlashLmpOn : Bool;
      CalcTime_FlashLmpOff : Time;
      CalcTime_FlashLmpOn : Time;
      R_Trig_StartShifting {InstructionName := 'R_TRIG'; LibVersion := '1.0'} : R_TRIG;
      Timer_ShiftingLight {InstructionName := 'TP_TIME'; LibVersion := '1.0'} : TP_TIME;
      F_TRIG_ShiftingLightOff {InstructionName := 'F_TRIG'; LibVersion := '1.0'} : F_TRIG;
      R_Edge_ShiftingLight { S7_SetPoint := 'True'} : Bool;
      F_Edge_TimerShiftingLight { S7_SetPoint := 'True'} : Bool;
      ShiftingLight : Byte;
   END_VAR


BEGIN
	
	REGION Flashing
	    // Stijgende flank om flashsignaal te activeren
	    #R_Trig_StartFlash(CLK := #iFlash,
	                       Q => #R_Edge_StartFlash);
	    // Tijd dat de lamp uit moet staan binnen een periode
	    #Timer_Flash_LmpOff(IN := #R_Edge_StartFlash OR #F_Edge_FlashLmpOn,
	                        PT := #CalcTime_FlashLmpOff);
	    // Dalende flank van deze gedoofde tijd
	    #F_TRIG_Flash_LmpOff(CLK := #Timer_Flash_LmpOff.Q,
	                         Q => #F_Edge_FlashLmpOff);
	    // Tijd dat de lamp aan moet staan binnen een periode
	    #Timer_Flash_LmpOn(IN := #R_Edge_StartFlash OR (#F_Edge_FlashLmpOff AND #iFlash),
	                       PT := #CalcTime_FlashLmpOn);
	    // Dalende flank van deze gedoofde tijd
	    #F_TRIG_Flash_LmpOn(CLK := #Timer_Flash_LmpOn.Q,
	                        Q => #F_Edge_FlashLmpOn);
	    
	    // Berekende tijd dat de lamp uit en aan moet staan binnen een periode
	    #CalcTime_FlashLmpOn := DINT_TO_TIME(REAL_TO_DINT((USINT_TO_REAL(#iSetting_Flash_Dutycycle) / 100.0 * #iSetting_Flash_Period) * 1000.0));
	    #CalcTime_FlashLmpOff :=DINT_TO_TIME(REAL_TO_DINT(#iSetting_Flash_Period * 1000.0)) - #CalcTime_FlashLmpOn;
	    
	    // Bij het uitzetten van iLmpFlash gaan we de timers resetten zodat het flashsignaal onmiddellijk dooft zonder zijn periode af te maken
	    IF NOT #iFlash
	    THEN
	        RESET_TIMER(#Timer_Flash_LmpOff);
	        RESET_TIMER(#Timer_Flash_LmpOn);
	    END_IF;
	END_REGION
	
	REGION Lamp
	    // Lamp continu of knipperend sturen
	    IF #iContinu
	    THEN
	        #oLmp := TRUE;
	    ELSE
	        #oLmp := #Timer_Flash_LmpOn.Q;
	    END_IF;
	END_REGION
	
	REGION ShiftingLight
	    // Stijgende flank om het looplicht te activeren
	    #R_Trig_StartShifting(CLK := #iShiftingLight,
	                         Q => #R_Edge_ShiftingLight);
	    // Dalende flank van timer die gebruikt wordt voor het looplicht
	    #F_TRIG_ShiftingLightOff(CLK:=#Timer_ShiftingLight.Q,
	                            Q=>#F_Edge_TimerShiftingLight);
	    // Tijd voor het opschuiven van het looplicht
	    #Timer_ShiftingLight(IN := #R_Edge_ShiftingLight OR #F_Edge_TimerShiftingLight,
	                        PT := DINT_TO_TIME(REAL_TO_DINT(#iSetting_ShiftInterval * 1000.0 )));
	    IF NOT #iShiftingLight
	    THEN
	        // Looplicht uit
	        #ShiftingLight := 0;
	    ELSIF #R_Edge_ShiftingLight 
	    THEN
	        // Set MSB van het looplicht
	        #ShiftingLight.%X7 := TRUE;
	    ELSIF #iShiftingLight AND #F_Edge_TimerShiftingLight
	    THEN
	        // Looplicht opschuiven
	        #ShiftingLight := ROR(IN := #ShiftingLight, N := 1);
	    END_IF;
	    #oShiftingLight := #ShiftingLight;
	END_REGION
	
END_FUNCTION_BLOCK

FUNCTION "FC_EM_Feeding" : Void   // FC2, FBD
TITLE = Feeding
{ S7_Optimized_Access := 'TRUE' }
// stored: SetENOAutomatically false
BEGIN

REGION Network 1: ------------------------------------------------------------------------ Inputs ------------------------------------------------------------------------
END_REGION

REGION Network 2: Verwerking iFeedingSenCilOut
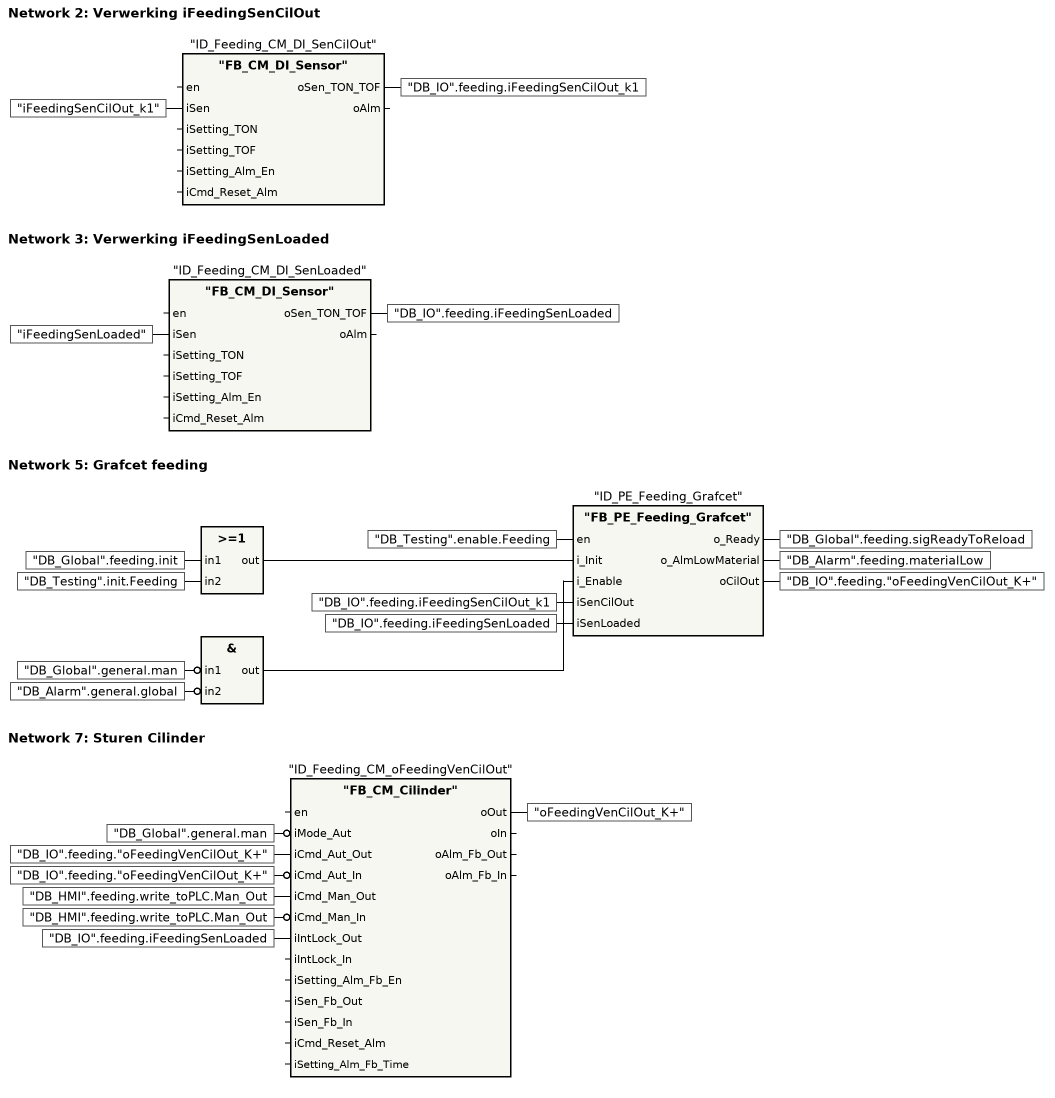
   "ID_Feeding_CM_DI_SenCilOut"(iSen := "iFeedingSenCilOut_k1",   // "FB_CM_DI_Sensor"
                           oSen_TON_TOF => "DB_IO".feeding.iFeedingSenCilOut_k1);
END_REGION

REGION Network 3: Verwerking iFeedingSenLoaded
   "ID_Feeding_CM_DI_SenLoaded"(iSen := "iFeedingSenLoaded", oSen_TON_TOF => "DB_IO".feeding.iFeedingSenLoaded);   // "FB_CM_DI_Sensor"
END_REGION

REGION Network 4: ------------------------------------------------------------------------ Logic ------------------------------------------------------------------------
END_REGION

REGION Network 5: Grafcet feeding
   IF "DB_Testing".enable.Feeding THEN
       "ID_PE_Feeding_Grafcet"(i_Init := "DB_Global".feeding.init OR "DB_Testing".init.Feeding,   // "FB_PE_Feeding_Grafcet"
                               i_Enable := NOT "DB_Global".general.man AND NOT "DB_Alarm".general.global,
                               iSenCilOut := "DB_IO".feeding.iFeedingSenCilOut_k1,
                               iSenLoaded := "DB_IO".feeding.iFeedingSenLoaded,
                               o_Ready => "DB_Global".feeding.sigReadyToReload,
                               o_AlmLowMaterial => "DB_Alarm".feeding.materialLow,
                               oCilOut => "DB_IO".feeding."oFeedingVenCilOut_K+");
   END_IF;
END_REGION

REGION Network 6: ------------------------------------------------------------------------ Outputs ------------------------------------------------------------------------
END_REGION

REGION Network 7: Sturen Cilinder
   "ID_Feeding_CM_oFeedingVenCilOut"(iMode_Aut := NOT "DB_Global".general.man,   // "FB_CM_Cilinder"
                           iCmd_Aut_Out := "DB_IO".feeding."oFeedingVenCilOut_K+",
                           iCmd_Aut_In := NOT "DB_IO".feeding."oFeedingVenCilOut_K+",
                           iCmd_Man_Out := "DB_HMI".feeding.write_toPLC.Man_Out,
                           iCmd_Man_In := NOT "DB_HMI".feeding.write_toPLC.Man_Out,
                           iIntLock_Out := "DB_IO".feeding.iFeedingSenLoaded,
                           oOut => "oFeedingVenCilOut_K+");
END_REGION
END_FUNCTION

FUNCTION_BLOCK "FB_PE_Feeding_Grafcet"
{ S7_Optimized_Access := 'TRUE' }
VERSION : 0.1
   VAR_INPUT 
      i_Init : Bool;
      i_Enable : Bool;
      iSenCilOut : Bool;
      iSenLoaded : Bool;
   END_VAR

   VAR_OUTPUT 
      o_Ready : Bool;
      o_AlmLowMaterial : Bool;
      oCilOut : Bool;
   END_VAR

   VAR 
      sStep : Int;
      sInit : Bool;
      sTON_X0 {InstructionName := 'TON_TIME'; LibVersion := '1.0'} : TON_TIME;
      sTON_X1 {InstructionName := 'TON_TIME'; LibVersion := '1.0'} : TON_TIME;
   END_VAR


BEGIN
	REGION init
	    IF #i_Init AND NOT (#sInit = #i_Init) THEN
	        #sStep := 0;
	    END_IF;
	    #sInit := #i_Init;
	END_REGION
	
	REGION Enable
	    IF NOT #i_Enable THEN
	        GOTO afterGrafcetLogic;
	    END_IF;
	END_REGION
	
	REGION Timers
	    
	    #sTON_X0(IN := NOT #iSenLoaded AND #sStep = 0,
	             PT := T#0.5S);
	    
	    #sTON_X1(IN := #iSenCilOut AND NOT #iSenLoaded AND #sStep = 1,
	                                PT := T#0.5S);
	    
	END_REGION
	
	REGION Grafcet logic
	    CASE #sStep OF
	        0: // o_Ready
	            IF #sTON_X0.Q THEN
	                #sStep := 1;
	            END_IF;
	        1: // oCilOut
	            IF #iSenCilOut AND #iSenLoaded THEN
	                #sStep := 0;
	            ELSIF #sTON_X1.Q THEN
	                #sStep := 2;
	            END_IF;
	        2: // o_AlmLowMaterial
	            ;
	        ELSE
	            #sStep := 0;
	    END_CASE;
	END_REGION
	
	afterGrafcetLogic: // Jump destination
	
	REGION Outputs
	    
	    #oCilOut := #sStep = 1;
	    #o_Ready := #sStep = 0;
	    #o_AlmLowMaterial := #sStep = 2;
	    
	END_REGION
END_FUNCTION_BLOCK

FUNCTION_BLOCK "FB_CM_Cilinder"   // FB1, FBD
TITLE = FB_CM_Cilinder AP BIB
{ S7_Optimized_Access := 'FALSE' }
// stored: SetENOAutomatically false
   VAR_INPUT
      iMode_Aut : Bool;
      iCmd_Aut_Out : Bool;
      iCmd_Aut_In : Bool;
      iCmd_Man_Out : Bool;
      iCmd_Man_In : Bool;
      iIntLock_Out : Bool;
      iIntLock_In : Bool;
      iSetting_Alm_Fb_En : Bool;
      iSen_Fb_Out : Bool;
      iSen_Fb_In : Bool;
      iCmd_Reset_Alm : Bool;
      iSetting_Alm_Fb_Time : Time;
   END_VAR
   VAR_OUTPUT
      oOut : Bool;
      oIn : Bool;
      oAlm_Fb_Out : Bool;
      oAlm_Fb_In : Bool;
   END_VAR
   VAR
      sHulpM : Array[0..15] of Bool;
      IEC_Timer_0_Instance { S7_SetPoint := 'True'} : TON_TIME;
      IEC_Timer_0_Instance_2 { S7_SetPoint := 'True'} : TON_TIME;
      s_iCmd_Auto_Out { S7_SetPoint := 'True'} : Bool;
      s_iCmd_Auto_In : Bool;
      s_iCmd_Man_Out_TRIG : Bool;
      s_iCmd_Man_In_TRIG : Bool;
   END_VAR
   VAR_TEMP   // added for the SCL form of the ladder/FBD networks
      _w1 : Bool;
   END_VAR
BEGIN

REGION Network 1: check input cmds in combination with mode and interlock
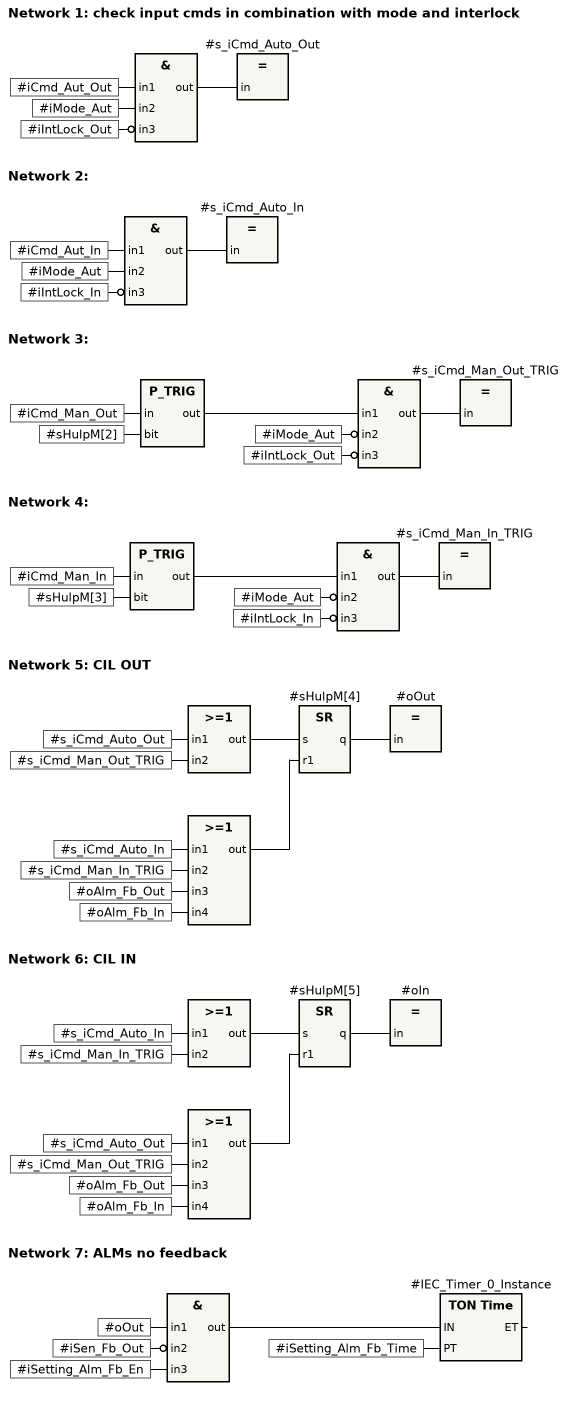
   #s_iCmd_Auto_Out := #iCmd_Aut_Out AND #iMode_Aut AND NOT #iIntLock_Out;
END_REGION

REGION Network 2
   #s_iCmd_Auto_In := #iCmd_Aut_In AND #iMode_Aut AND NOT #iIntLock_In;
END_REGION

REGION Network 3
   #_w1 := #iCmd_Man_Out AND NOT #sHulpM[2];   // rising edge
   #sHulpM[2] := #iCmd_Man_Out;
   #s_iCmd_Man_Out_TRIG := #_w1 AND NOT #iMode_Aut AND NOT #iIntLock_Out;
END_REGION

REGION Network 4
   #_w1 := #iCmd_Man_In AND NOT #sHulpM[3];   // rising edge
   #sHulpM[3] := #iCmd_Man_In;
   #s_iCmd_Man_In_TRIG := #_w1 AND NOT #iMode_Aut AND NOT #iIntLock_In;
END_REGION

REGION Network 5: CIL OUT
   // SET cilinder out: auto or man out command
   // 
   // RESET cilinder out: auto or man in command or alarm
   IF #s_iCmd_Auto_Out OR #s_iCmd_Man_Out_TRIG THEN
       #sHulpM[4] := TRUE;   // SR flip-flop
   END_IF;
   IF #s_iCmd_Auto_In OR #s_iCmd_Man_In_TRIG OR #oAlm_Fb_Out OR #oAlm_Fb_In THEN #sHulpM[4] := FALSE; END_IF;
   #oOut := #sHulpM[4];
END_REGION

REGION Network 6: CIL IN
   // SET cilinder in: auto or man in command
   // 
   // RESET cilinder in: auto or man out command or alarm
   IF #s_iCmd_Auto_In OR #s_iCmd_Man_In_TRIG THEN
       #sHulpM[5] := TRUE;   // SR flip-flop
   END_IF;
   IF #s_iCmd_Auto_Out OR #s_iCmd_Man_Out_TRIG OR #oAlm_Fb_Out OR #oAlm_Fb_In THEN
       #sHulpM[5] := FALSE;
   END_IF;
   #oIn := #sHulpM[5];
END_REGION

REGION Network 7: ALMs no feedback
   #IEC_Timer_0_Instance(IN := #oOut AND NOT #iSen_Fb_Out AND #iSetting_Alm_Fb_En, PT := #iSetting_Alm_Fb_Time);   // TON
END_REGION

REGION Network 8
   // om compatibel te zijn met 300-PLC, mag er niets achter de TON worden geprogrammeerd
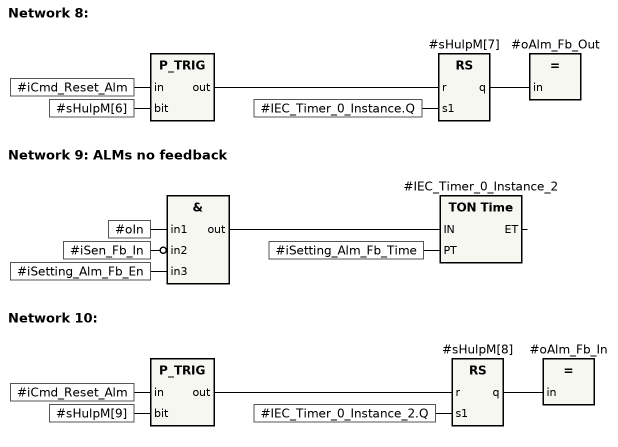
   #_w1 := #iCmd_Reset_Alm AND NOT #sHulpM[6];   // rising edge
   #sHulpM[6] := #iCmd_Reset_Alm;
   IF #_w1 THEN
       #sHulpM[7] := FALSE;   // RS flip-flop
   END_IF;
   IF #IEC_Timer_0_Instance.Q THEN #sHulpM[7] := TRUE; END_IF;
   #oAlm_Fb_Out := #sHulpM[7];
END_REGION

REGION Network 9: ALMs no feedback
   #IEC_Timer_0_Instance_2(IN := #oIn AND NOT #iSen_Fb_In AND #iSetting_Alm_Fb_En, PT := #iSetting_Alm_Fb_Time);   // TON
END_REGION

REGION Network 10
   #_w1 := #iCmd_Reset_Alm AND NOT #sHulpM[9];   // rising edge
   #sHulpM[9] := #iCmd_Reset_Alm;
   IF #_w1 THEN
       #sHulpM[8] := FALSE;   // RS flip-flop
   END_IF;
   IF #IEC_Timer_0_Instance_2.Q THEN #sHulpM[8] := TRUE; END_IF;
   #oAlm_Fb_In := #sHulpM[8];
END_REGION

REGION Network 11: statusword TODO
END_REGION
END_FUNCTION_BLOCK

FUNCTION "FC_EM_Loading" : Void   // FC3, FBD
{ S7_Optimized_Access := 'TRUE' }
// stored: SetENOAutomatically false
BEGIN

REGION Network 1: ------------------------------------------------------------------------ Inputs ------------------------------------------------------------------------
END_REGION

REGION Network 2: Verwerken iLoadingSenDown_a1
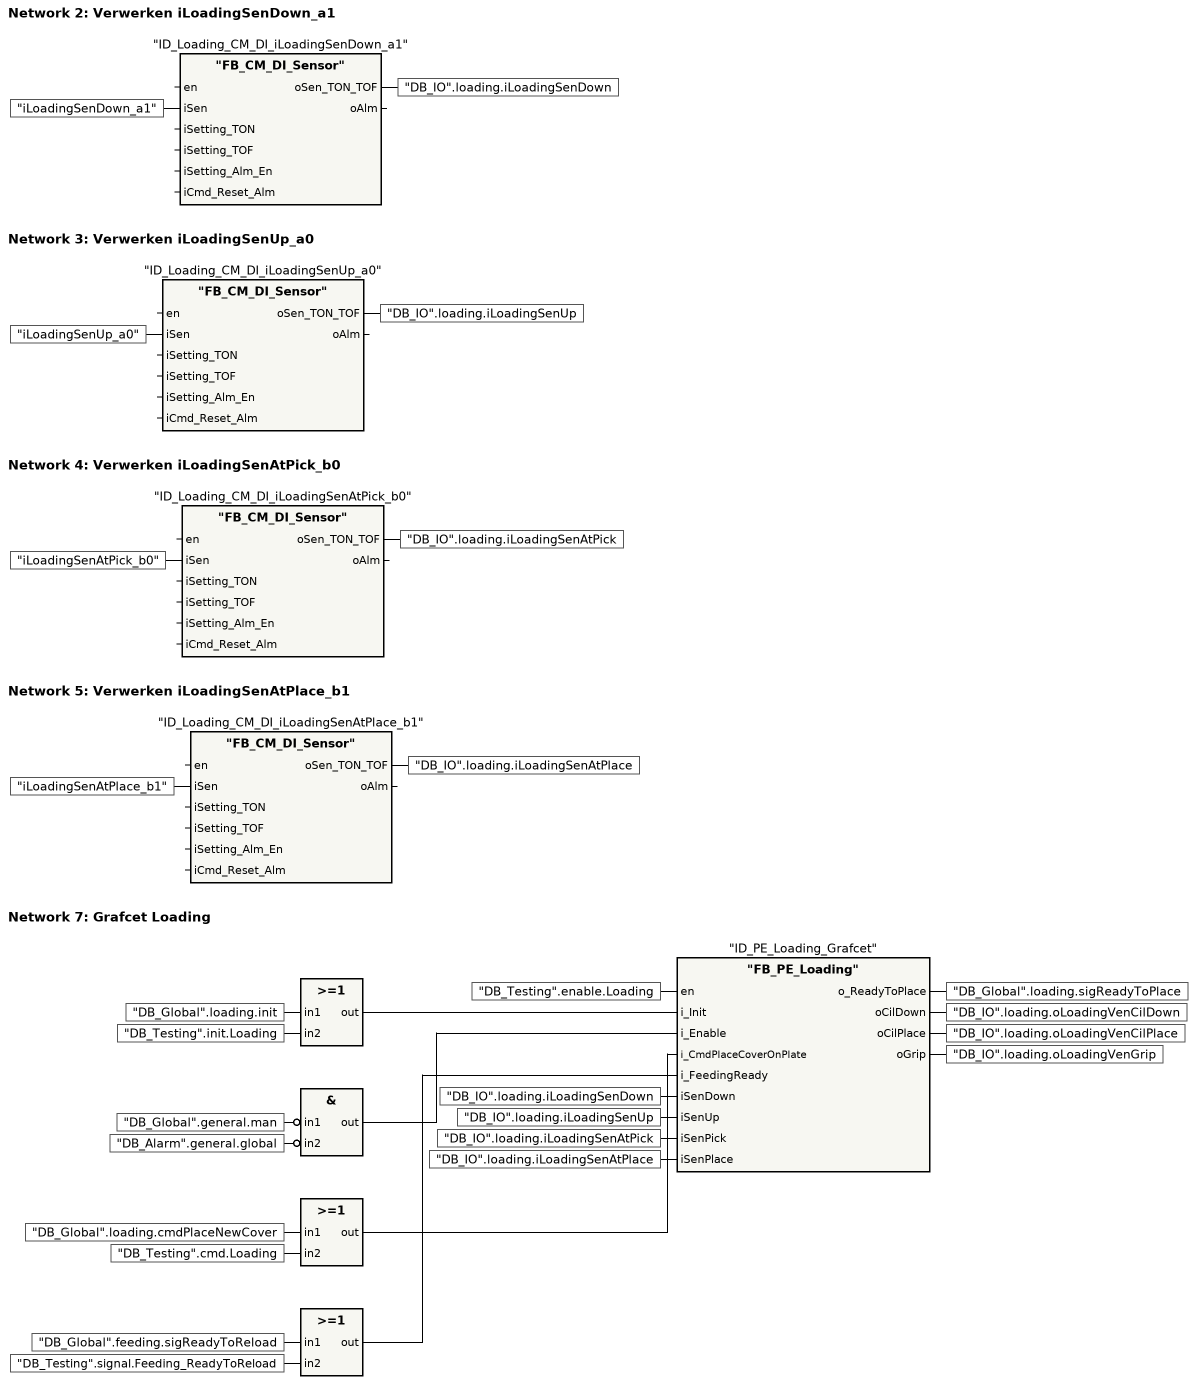
   "ID_Loading_CM_DI_iLoadingSenDown_a1"(iSen := "iLoadingSenDown_a1",   // "FB_CM_DI_Sensor"
                           oSen_TON_TOF => "DB_IO".loading.iLoadingSenDown);
END_REGION

REGION Network 3: Verwerken iLoadingSenUp_a0
   "ID_Loading_CM_DI_iLoadingSenUp_a0"(iSen := "iLoadingSenUp_a0",   // "FB_CM_DI_Sensor"
                           oSen_TON_TOF => "DB_IO".loading.iLoadingSenUp);
END_REGION

REGION Network 4: Verwerken iLoadingSenAtPick_b0
   "ID_Loading_CM_DI_iLoadingSenAtPick_b0"(iSen := "iLoadingSenAtPick_b0",   // "FB_CM_DI_Sensor"
                           oSen_TON_TOF => "DB_IO".loading.iLoadingSenAtPick);
END_REGION

REGION Network 5: Verwerken iLoadingSenAtPlace_b1
   "ID_Loading_CM_DI_iLoadingSenAtPlace_b1"(iSen := "iLoadingSenAtPlace_b1",   // "FB_CM_DI_Sensor"
                           oSen_TON_TOF => "DB_IO".loading.iLoadingSenAtPlace);
END_REGION

REGION Network 6: ------------------------------------------------------------------------ Logic ------------------------------------------------------------------------
END_REGION

REGION Network 7: Grafcet Loading
   IF "DB_Testing".enable.Loading THEN
       "ID_PE_Loading_Grafcet"(i_Init := "DB_Global".loading.init OR "DB_Testing".init.Loading,   // "FB_PE_Loading"
                               i_Enable := NOT "DB_Global".general.man AND NOT "DB_Alarm".general.global,
                               i_CmdPlaceCoverOnPlate := "DB_Global".loading.cmdPlaceNewCover OR "DB_Testing".cmd.Loading,
                               i_FeedingReady := "DB_Global".feeding.sigReadyToReload OR "DB_Testing".signal.Feeding_ReadyToReload,
                               iSenDown := "DB_IO".loading.iLoadingSenDown,
                               iSenUp := "DB_IO".loading.iLoadingSenUp,
                               iSenPick := "DB_IO".loading.iLoadingSenAtPick,
                               iSenPlace := "DB_IO".loading.iLoadingSenAtPlace,
                               o_ReadyToPlace => "DB_Global".loading.sigReadyToPlace,
                               oCilDown => "DB_IO".loading.oLoadingVenCilDown,
                               oCilPlace => "DB_IO".loading.oLoadingVenCilPlace,
                               oGrip => "DB_IO".loading.oLoadingVenGrip);
   END_IF;
END_REGION

REGION Network 8: ------------------------------------------------------------------------ Outputs ------------------------------------------------------------------------
END_REGION

REGION Network 9: Sturen oLoadingVenCilDown_A+
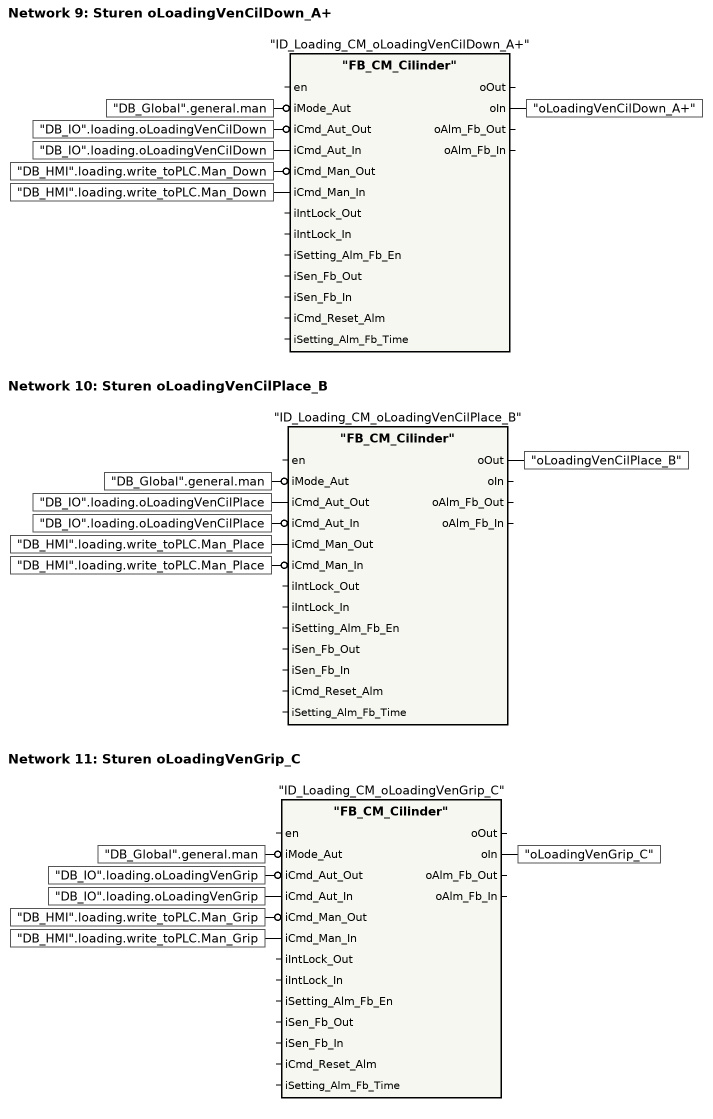
   "ID_Loading_CM_oLoadingVenCilDown_A+"(iMode_Aut := NOT "DB_Global".general.man,   // "FB_CM_Cilinder"
                           iCmd_Aut_Out := NOT "DB_IO".loading.oLoadingVenCilDown,
                           iCmd_Aut_In := "DB_IO".loading.oLoadingVenCilDown,
                           iCmd_Man_Out := NOT "DB_HMI".loading.write_toPLC.Man_Down,
                           iCmd_Man_In := "DB_HMI".loading.write_toPLC.Man_Down,
                           oIn => "oLoadingVenCilDown_A+");
END_REGION

REGION Network 10: Sturen oLoadingVenCilPlace_B
   "ID_Loading_CM_oLoadingVenCilPlace_B"(iMode_Aut := NOT "DB_Global".general.man,   // "FB_CM_Cilinder"
                           iCmd_Aut_Out := "DB_IO".loading.oLoadingVenCilPlace,
                           iCmd_Aut_In := NOT "DB_IO".loading.oLoadingVenCilPlace,
                           iCmd_Man_Out := "DB_HMI".loading.write_toPLC.Man_Place,
                           iCmd_Man_In := NOT "DB_HMI".loading.write_toPLC.Man_Place,
                           oOut => "oLoadingVenCilPlace_B");
END_REGION

REGION Network 11: Sturen oLoadingVenGrip_C
   "ID_Loading_CM_oLoadingVenGrip_C"(iMode_Aut := NOT "DB_Global".general.man,   // "FB_CM_Cilinder"
                           iCmd_Aut_Out := NOT "DB_IO".loading.oLoadingVenGrip,
                           iCmd_Aut_In := "DB_IO".loading.oLoadingVenGrip,
                           iCmd_Man_Out := NOT "DB_HMI".loading.write_toPLC.Man_Grip,
                           iCmd_Man_In := "DB_HMI".loading.write_toPLC.Man_Grip,
                           oIn => "oLoadingVenGrip_C");
END_REGION
END_FUNCTION

FUNCTION_BLOCK "FB_PE_Loading"
{ S7_Optimized_Access := 'TRUE' }
VERSION : 0.1
   VAR_INPUT 
      i_Init : Bool;
      i_Enable : Bool;
      i_CmdPlaceCoverOnPlate : Bool;
      i_FeedingReady : Bool;
      iSenDown : Bool;
      iSenUp : Bool;
      iSenPick : Bool;
      iSenPlace : Bool;
   END_VAR

   VAR_OUTPUT 
      o_ReadyToPlace : Bool;
      oCilDown : Bool;
      oCilPlace : Bool;
      oGrip : Bool;
   END_VAR

   VAR 
      sStep : Int;
      sInit : Bool;
      sTON_X1 {InstructionName := 'TON_TIME'; LibVersion := '1.0'} : TON_TIME;
      sTON_X2 {InstructionName := 'TON_TIME'; LibVersion := '1.0'} : TON_TIME;
      sTON_X3 {InstructionName := 'TON_TIME'; LibVersion := '1.0'} : TON_TIME;
      sTON_X4 {InstructionName := 'TON_TIME'; LibVersion := '1.0'} : TON_TIME;
      sTON_X5 {InstructionName := 'TON_TIME'; LibVersion := '1.0'} : TON_TIME;
      sTON_X6 {InstructionName := 'TON_TIME'; LibVersion := '1.0'} : TON_TIME;
   END_VAR

   VAR CONSTANT 
      c_time : Time := T#0.5s;
   END_VAR


BEGIN
	REGION init
	    IF #i_Init AND NOT (#sInit = #i_Init) THEN
	        #sStep := 0;
	    END_IF;
	    #sInit := #i_Init;
	END_REGION
	
	REGION Enable
	    IF NOT #i_Enable THEN
	        GOTO afterGrafcetLogic;
	    END_IF;
	END_REGION
	
	REGION Timers
	    
	    #sTON_X1(
	        IN:= #sStep = 1 AND #iSenDown,
	        PT:=#c_time
	    );
	    
	    #sTON_X2(
	        IN:= #sStep = 2,
	        PT:= #c_time
	    );
	    
	    #sTON_X3(
	        IN:= #sStep = 3 AND #iSenUp,
	        PT:= #c_time
	    );
	    
	    #sTON_X4(
	        IN:= #sStep = 4 AND #iSenPlace,
	        PT:= #c_time
	    );
	    
	    #sTON_X5(
	        IN:= #sStep = 5 AND #iSenDown,
	        PT:= #c_time
	    );
	    
	    #sTON_X6(
	        IN:= #sStep = 6,
	        PT:= #c_time
	    );
	    
	END_REGION
	
	REGION Grafcet logic
	    CASE #sStep OF
	        0:
	            IF #i_FeedingReady AND #iSenPick  AND #i_CmdPlaceCoverOnPlate AND #iSenUp THEN
	                #sStep := 1;
	            END_IF;
	        1:
	            IF #sTON_X1.Q THEN
	                #sStep := 2;
	            END_IF;
	        2:
	            IF #sTON_X2.Q THEN
	                #sStep := 3;
	            END_IF;
	        3:
	            IF #sTON_X3.Q THEN
	                #sStep := 4;
	            END_IF;
	        4:
	            IF #sTON_X4.Q THEN
	                #sStep := 5;
	            END_IF;
	        5:
	            IF #sTON_X5.Q THEN
	                #sStep := 6;
	            END_IF;
	        6:
	            IF #sTON_X6.Q THEN
	                #sStep := 7;
	            END_IF;
	        7:
	            IF #iSenUp THEN
	                #sStep := 0;
	            END_IF;
	        ELSE  // Statement section ELSE
	            #sStep := 0;
	    END_CASE;
	END_REGION
	
	afterGrafcetLogic: // Jump destination
	
	REGION Outputs
	    
	    #o_ReadyToPlace := #sStep = 0;
	    #oCilDown := #sStep = 1 OR #sStep = 2 OR #sStep = 5 OR #sStep = 6;
	    #oCilPlace := #sStep = 4 OR #sStep = 5 OR #sStep = 6 OR #sStep = 7;
	    #oGrip := #sStep = 2 OR #sStep = 3 OR #sStep = 4 OR #sStep = 5;
	    
	END_REGION
END_FUNCTION_BLOCK

FUNCTION "FC_EM_Plate" : Void   // FC4, FBD
{ S7_Optimized_Access := 'TRUE' }
// stored: SetENOAutomatically false
   VAR_TEMP
      Debug : Bool;
   END_VAR
BEGIN

REGION Network 1: ------------------------------------------------------------------------ Inputs ------------------------------------------------------------------------
END_REGION

REGION Network 2: Verwerken iPlateSenCilPushingIn_d0
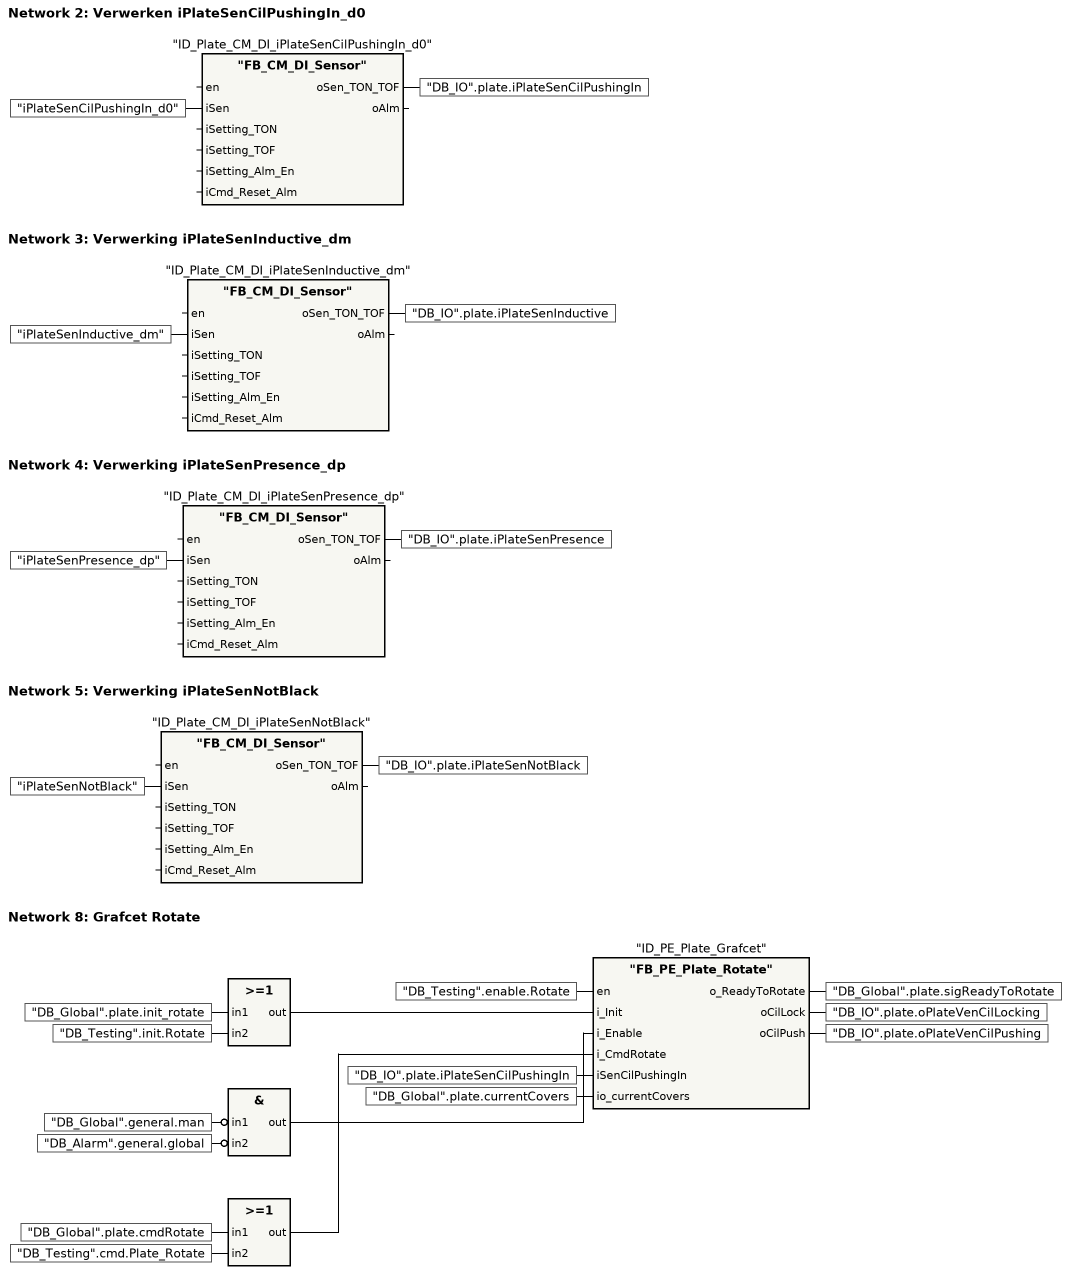
   "ID_Plate_CM_DI_iPlateSenCilPushingIn_d0"(iSen := "iPlateSenCilPushingIn_d0",   // "FB_CM_DI_Sensor"
                           oSen_TON_TOF => "DB_IO".plate.iPlateSenCilPushingIn);
END_REGION

REGION Network 3: Verwerking iPlateSenInductive_dm
   "ID_Plate_CM_DI_iPlateSenInductive_dm"(iSen := "iPlateSenInductive_dm",   // "FB_CM_DI_Sensor"
                           oSen_TON_TOF => "DB_IO".plate.iPlateSenInductive);
END_REGION

REGION Network 4: Verwerking iPlateSenPresence_dp
   "ID_Plate_CM_DI_iPlateSenPresence_dp"(iSen := "iPlateSenPresence_dp",   // "FB_CM_DI_Sensor"
                           oSen_TON_TOF => "DB_IO".plate.iPlateSenPresence);
END_REGION

REGION Network 5: Verwerking iPlateSenNotBlack
   "ID_Plate_CM_DI_iPlateSenNotBlack"(iSen := "iPlateSenNotBlack",   // "FB_CM_DI_Sensor"
                           oSen_TON_TOF => "DB_IO".plate.iPlateSenNotBlack);
END_REGION

REGION Network 6 (SCL): Verwerking iPlateSenHeight
   "DB_IO".plate.iPlateSenHeight := "iPlateSenHeight";
END_REGION

REGION Network 7: ------------------------------------------------------------------------ Logic ------------------------------------------------------------------------
END_REGION

REGION Network 8: Grafcet Rotate
   IF "DB_Testing".enable.Rotate THEN
       "ID_PE_Plate_Grafcet"(i_Init := "DB_Global".plate.init_rotate OR "DB_Testing".init.Rotate,   // "FB_PE_Plate_Rotate"
                             i_Enable := NOT "DB_Global".general.man AND NOT "DB_Alarm".general.global,
                             i_CmdRotate := "DB_Global".plate.cmdRotate OR "DB_Testing".cmd.Plate_Rotate,
                             iSenCilPushingIn := "DB_IO".plate.iPlateSenCilPushingIn,
                             io_currentCovers := "DB_Global".plate.currentCovers,
                             o_ReadyToRotate => "DB_Global".plate.sigReadyToRotate,
                             oCilLock => "DB_IO".plate.oPlateVenCilLocking,
                             oCilPush => "DB_IO".plate.oPlateVenCilPushing);
   END_IF;
END_REGION

REGION Network 9: Grafcet Measure
   // TODO:
   // - Correct placement in array
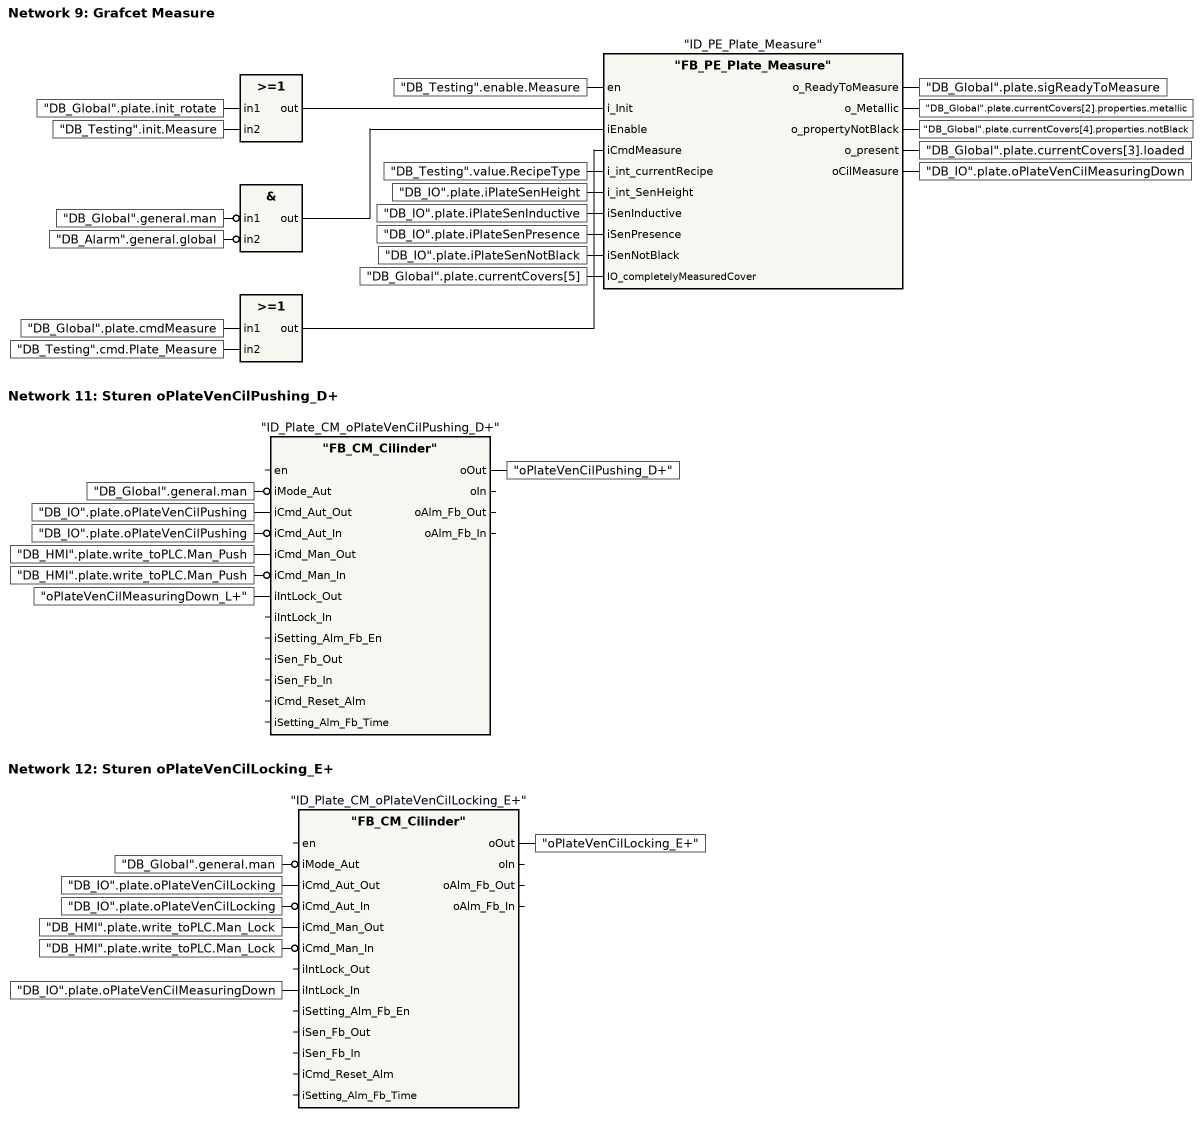
   IF "DB_Testing".enable.Measure THEN
       "ID_PE_Plate_Measure"(i_Init := "DB_Global".plate.init_rotate OR "DB_Testing".init.Measure,   // "FB_PE_Plate_Measure"
                             iEnable := NOT "DB_Global".general.man AND NOT "DB_Alarm".general.global,
                             iCmdMeasure := "DB_Global".plate.cmdMeasure OR "DB_Testing".cmd.Plate_Measure,
                             i_int_currentRecipe := "DB_Testing".value.RecipeType,
                             i_int_SenHeight := "DB_IO".plate.iPlateSenHeight,
                             iSenInductive := "DB_IO".plate.iPlateSenInductive,
                             iSenPresence := "DB_IO".plate.iPlateSenPresence,
                             iSenNotBlack := "DB_IO".plate.iPlateSenNotBlack,
                             IO_completelyMeasuredCover := "DB_Global".plate.currentCovers[5],
                             o_ReadyToMeasure => "DB_Global".plate.sigReadyToMeasure,
                             o_Metallic => "DB_Global".plate.currentCovers[2].properties.metallic,
                             o_propertyNotBlack => "DB_Global".plate.currentCovers[4].properties.notBlack,
                             o_present => "DB_Global".plate.currentCovers[3].loaded,
                             oCilMeasure => "DB_IO".plate.oPlateVenCilMeasuringDown);
   END_IF;
END_REGION

REGION Network 10: ------------------------------------------------------------------------ Outputs ------------------------------------------------------------------------
END_REGION

REGION Network 11: Sturen oPlateVenCilPushing_D+
   "ID_Plate_CM_oPlateVenCilPushing_D+"(iMode_Aut := NOT "DB_Global".general.man,   // "FB_CM_Cilinder"
                           iCmd_Aut_Out := "DB_IO".plate.oPlateVenCilPushing,
                           iCmd_Aut_In := NOT "DB_IO".plate.oPlateVenCilPushing,
                           iCmd_Man_Out := "DB_HMI".plate.write_toPLC.Man_Push,
                           iCmd_Man_In := NOT "DB_HMI".plate.write_toPLC.Man_Push,
                           iIntLock_Out := "oPlateVenCilMeasuringDown_L+",
                           oOut => "oPlateVenCilPushing_D+");
END_REGION

REGION Network 12: Sturen oPlateVenCilLocking_E+
   "ID_Plate_CM_oPlateVenCilLocking_E+"(iMode_Aut := NOT "DB_Global".general.man,   // "FB_CM_Cilinder"
                           iCmd_Aut_Out := "DB_IO".plate.oPlateVenCilLocking,
                           iCmd_Aut_In := NOT "DB_IO".plate.oPlateVenCilLocking,
                           iCmd_Man_Out := "DB_HMI".plate.write_toPLC.Man_Lock,
                           iCmd_Man_In := NOT "DB_HMI".plate.write_toPLC.Man_Lock,
                           iIntLock_In := "DB_IO".plate.oPlateVenCilMeasuringDown,
                           oOut => "oPlateVenCilLocking_E+");
END_REGION

REGION Network 13: Sturen oPlateVenCilMeasuringDown_L+
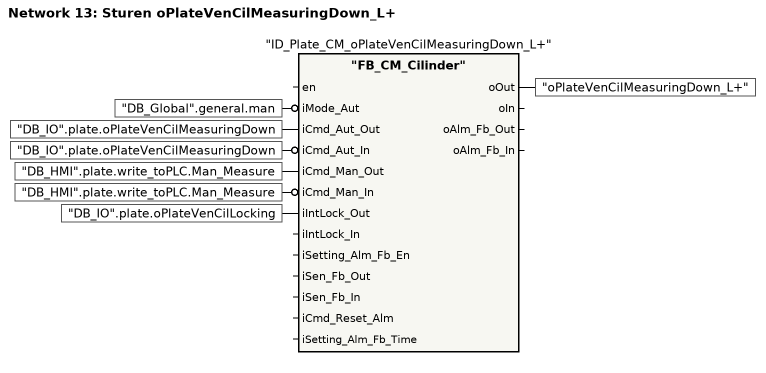
   "ID_Plate_CM_oPlateVenCilMeasuringDown_L+"(iMode_Aut := NOT "DB_Global".general.man,   // "FB_CM_Cilinder"
                           iCmd_Aut_Out := "DB_IO".plate.oPlateVenCilMeasuringDown,
                           iCmd_Aut_In := NOT "DB_IO".plate.oPlateVenCilMeasuringDown,
                           iCmd_Man_Out := "DB_HMI".plate.write_toPLC.Man_Measure,
                           iCmd_Man_In := NOT "DB_HMI".plate.write_toPLC.Man_Measure,
                           iIntLock_Out := "DB_IO".plate.oPlateVenCilLocking,
                           oOut => "oPlateVenCilMeasuringDown_L+");
END_REGION
END_FUNCTION

FUNCTION_BLOCK "FB_PE_Plate_Rotate"
{ S7_Optimized_Access := 'TRUE' }
VERSION : 0.1
   VAR_INPUT 
      i_Init : Bool;
      i_Enable : Bool;
      i_CmdRotate : Bool;
      iSenCilPushingIn : Bool;
   END_VAR

   VAR_OUTPUT 
      o_ReadyToRotate : Bool;
      oCilLock : Bool;
      oCilPush : Bool;
   END_VAR

   VAR_IN_OUT 
      io_currentCovers : Array[0..7] of "UDT_coverProperties";
   END_VAR

   VAR 
      sStep : Int;
      sInit : Bool;
      sTON_X1 {InstructionName := 'TON_TIME'; LibVersion := '1.0'} : TON_TIME;
      sTON_X2 {InstructionName := 'TON_TIME'; LibVersion := '1.0'} : TON_TIME;
      sTON_X3 {InstructionName := 'TON_TIME'; LibVersion := '1.0'} : TON_TIME;
   END_VAR

   VAR_TEMP 
      x_currentCovers : Array[0..7] of "UDT_coverProperties";
      x_lastCover : "UDT_coverProperties";
      i : Int;
   END_VAR

   VAR CONSTANT 
      c_time : Time := T#0.5s;
   END_VAR


BEGIN
	REGION init
	    IF #i_Init AND NOT (#sInit = #i_Init) THEN
	        #sStep := 0;
	    END_IF;
	    #sInit := #i_Init;
	END_REGION
	
	REGION enable
	    IF NOT #i_Enable THEN
	        GOTO afterGrafcetLogic;
	    END_IF;
	END_REGION
	
	REGION timers
	    #sTON_X1(IN := #sStep = 1,
	                  PT := #c_time);
	    
	    #sTON_X2(IN := #sStep = 2,
	                  PT := #c_time);
	    
	    #sTON_X3(IN := #sStep = 3,
	                  PT := #c_time);
	END_REGION
	
	REGION grafcet logic
	    CASE #sStep OF
	        0:
	            IF #i_CmdRotate AND #iSenCilPushingIn THEN
	                #sStep := 1;
	            END_IF;
	        1:
	            IF #sTON_X1.Q THEN
	                #sStep := 2;
	            END_IF;
	        2:
	            IF #sTON_X2.Q THEN
	                #sStep := 3;
	            END_IF;
	        3:
	            #sStep := 4;
	        4:
	            IF #sTON_X3.Q THEN
	                #sStep := 0;
	            END_IF;
	        ELSE
	            #sStep := 0;
	    END_CASE;
	END_REGION
	
	afterGrafcetLogic: // Jump destination
	
	REGION rotate array
	    
	    IF #sStep = 3 THEN
	        #x_currentCovers := #io_currentCovers; // Write to temp
	        #x_lastCover := #x_currentCovers[7]; // Save last in temp
	        
	        FOR #i := 7 TO 1 BY -1 DO
	            // Rotate array
	            #x_currentCovers[#i] := #x_currentCovers[#i - 1];
	        END_FOR;
	        #x_currentCovers[0] := #x_lastCover; // Set first to last in temp
	        
	        #io_currentCovers := #x_currentCovers; // Output
	    END_IF;
	    
	END_REGION
	
	REGION outputs
	    
	    #o_ReadyToRotate := #sStep = 0;
	    #oCilLock := #sStep = 1 OR #sStep = 2;
	    #oCilPush := #sStep = 2 OR #sStep = 3;
	    
	END_REGION
	    
END_FUNCTION_BLOCK

FUNCTION_BLOCK "FB_PE_Plate_Measure"
{ S7_Optimized_Access := 'TRUE' }
VERSION : 0.1
   VAR_INPUT 
      i_Init : Bool;
      iEnable : Bool;
      iCmdMeasure : Bool;
      i_int_currentRecipe : Int;
      i_int_SenHeight : Int;
      iSenInductive : Bool;
      iSenPresence : Bool;
      iSenNotBlack : Bool;
   END_VAR

   VAR_OUTPUT 
      o_ReadyToMeasure : Bool;
      o_Metallic : Bool;
      o_propertyNotBlack : Bool;
      o_present : Bool;
      oCilMeasure : Bool;
   END_VAR

   VAR_IN_OUT 
      IO_completelyMeasuredCover : "UDT_coverProperties";
   END_VAR

   VAR 
      sStep : Int;
      sInit : Bool;
      s_int_Previous : Int;
      sTON_X1 {InstructionName := 'TON_TIME'; LibVersion := '1.0'} : TON_TIME;
      sTON_X3 {InstructionName := 'TON_TIME'; LibVersion := '1.0'} : TON_TIME;
   END_VAR

   VAR CONSTANT 
      c_time_WaitTime : Time := T#0.5s;
      c_int_MaxMeasureForOk : Int := 1590;
   END_VAR


BEGIN
	REGION init
	    IF #i_Init AND NOT (#sInit = #i_Init) THEN
	        #sStep := 0;
	    END_IF;
	    #sInit := #i_Init;
	END_REGION
	
	REGION enable
	    IF NOT #iEnable THEN
	        GOTO afterGrafcetLogic;
	    END_IF;
	END_REGION
	
	REGION timers
	    
	    #sTON_X1(IN:= #s_int_Previous = #i_int_SenHeight,
	             PT:= #c_time_WaitTime);
	
	    #sTON_X3(IN:= #i_int_SenHeight < 20,
	             PT:= #c_time_WaitTime);
	    
	END_REGION
	
	REGION grafcet logic
	    CASE #sStep OF
	        0:
	            IF #iCmdMeasure THEN
	                #sStep := 1;
	            END_IF;
	        1:
	            IF #sTON_X1.Q THEN
	                #sStep := 2;
	            END_IF;
	        2:
	            #sStep := 3;
	        3:
	            IF #sTON_X3.Q THEN
	                #sStep := 0;
	            END_IF;
	        ELSE
	            #sStep := 0;
	    END_CASE;
	END_REGION
	
	afterGrafcetLogic: // Jump destination
	
	REGION outputs
	    #o_ReadyToMeasure := #sStep = 0;
	    #oCilMeasure := #sStep = 1;
	    
	    IF #sStep = 2 THEN
	        #o_Metallic := #iSenInductive;
	        #o_propertyNotBlack := #iSenNotBlack;
	        #o_present := #iSenPresence;
	        
	        IF (#i_int_SenHeight < #"c_int_MaxMeasureForOk") THEN
	            #IO_completelyMeasuredCover.properties.correctOrientation := TRUE;
	        ELSE
	            #IO_completelyMeasuredCover.properties.correctOrientation := FALSE;
	        END_IF;
	        
	        #IO_completelyMeasuredCover.reject := "FC_setRejectBitInCoverProperties"( i_currentCover := #IO_completelyMeasuredCover, i_currentRecipe := #i_int_currentRecipe);
	    END_IF;
	END_REGION
	
	REGION set static mem
	    #s_int_Previous := #i_int_SenHeight;
	END_REGION
	    
END_FUNCTION_BLOCK

FUNCTION "FC_setRejectBitInCoverProperties" : Bool
{ S7_Optimized_Access := 'TRUE' }
VERSION : 0.1
   VAR_INPUT 
      i_currentCover : "UDT_coverProperties";
      i_currentRecipe : Int;
   END_VAR


BEGIN
	REGION Don't reject empty place
	    IF
	        NOT #i_currentCover.loaded
	    THEN
	        #FC_setRejectBitInCoverProperties := FALSE;
	        RETURN;
	    END_IF;
	END_REGION
	
	REGION Check recipe
	    
	    // Recipe
	    // 1 = Black
	    // 2 = Metallic
	    
	    REGION Black
	        IF
	            (#i_currentRecipe = 1)
	            AND NOT (#i_currentCover.properties.metallic)
	            AND NOT (#i_currentCover.properties.notBlack)
	        THEN
	            #FC_setRejectBitInCoverProperties := FALSE;
	            RETURN;
	        END_IF;
	    END_REGION
	    
	    REGION Metallic
	        IF
	            (#i_currentRecipe = 2)
	            AND #i_currentCover.properties.metallic
	        THEN
	            #FC_setRejectBitInCoverProperties := FALSE;
	            RETURN;
	        END_IF;
	    END_REGION
	END_REGION
	
	#FC_setRejectBitInCoverProperties := TRUE;
END_FUNCTION

FUNCTION "FC_EM_Reject" : Void   // FC5, FBD
{ S7_Optimized_Access := 'TRUE' }
// stored: SetENOAutomatically false
BEGIN

REGION Network 1: ------------------------------------------------------------------------ Inputs ------------------------------------------------------------------------
END_REGION

REGION Network 2: Verwerking iRejectSenCilIn_f0
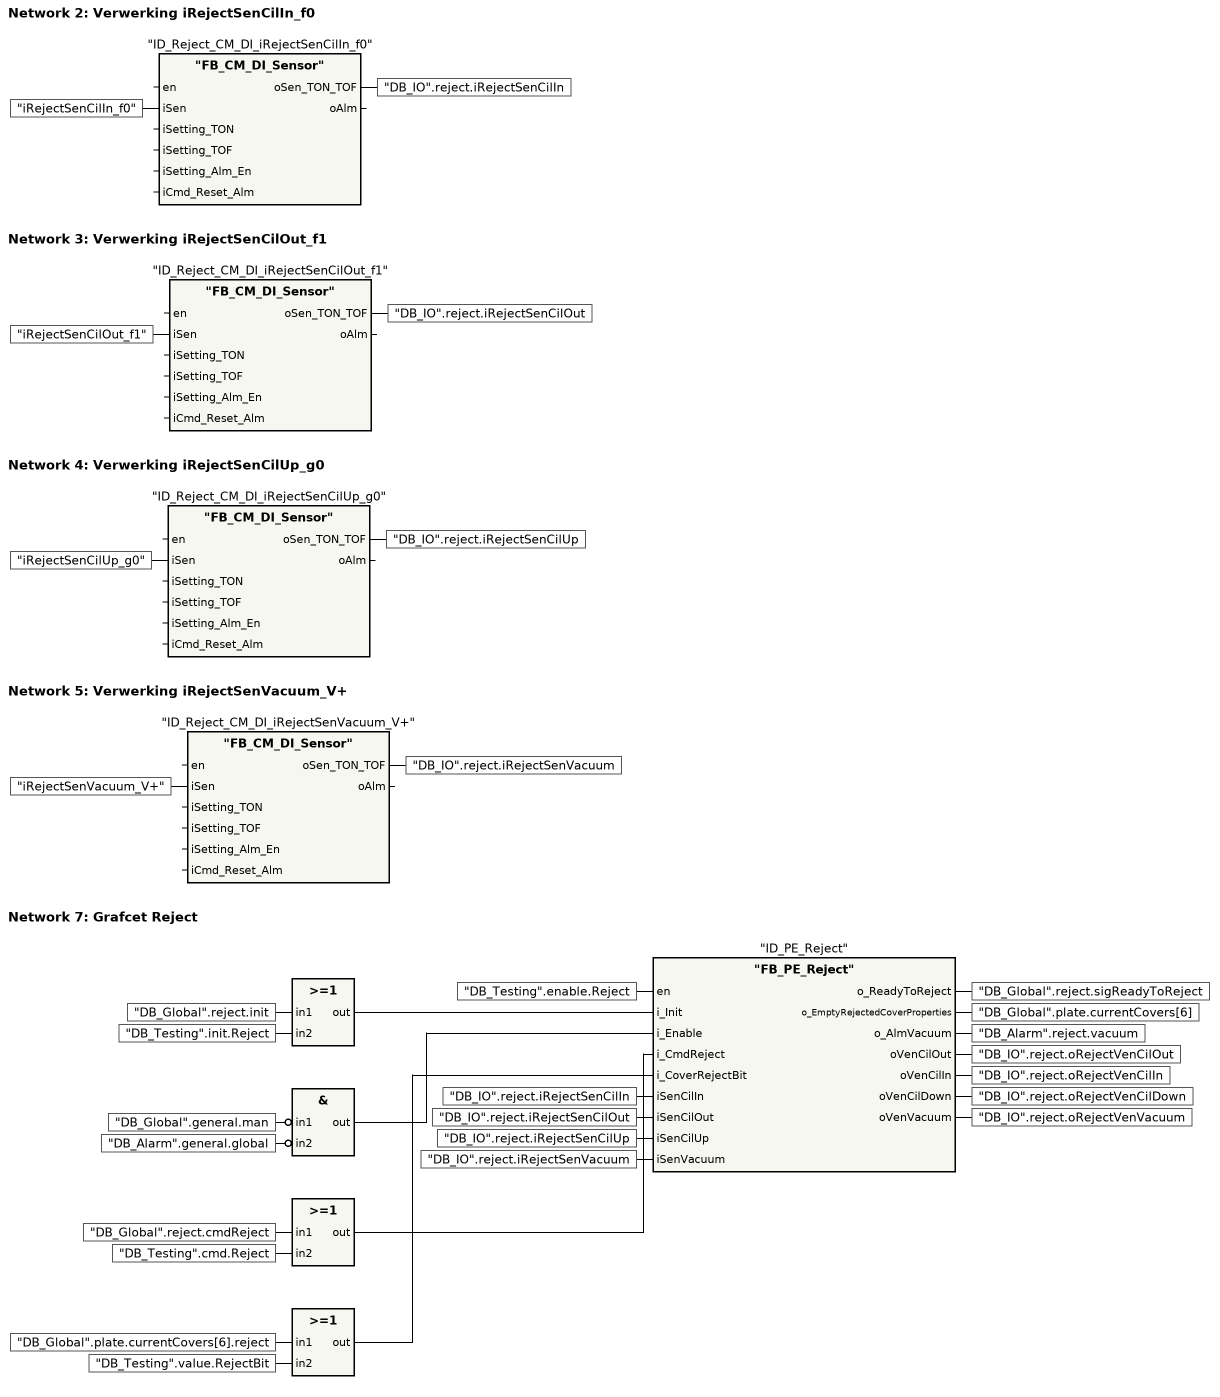
   "ID_Reject_CM_DI_iRejectSenCilIn_f0"(iSen := "iRejectSenCilIn_f0",   // "FB_CM_DI_Sensor"
                           oSen_TON_TOF => "DB_IO".reject.iRejectSenCilIn);
END_REGION

REGION Network 3: Verwerking iRejectSenCilOut_f1
   "ID_Reject_CM_DI_iRejectSenCilOut_f1"(iSen := "iRejectSenCilOut_f1",   // "FB_CM_DI_Sensor"
                           oSen_TON_TOF => "DB_IO".reject.iRejectSenCilOut);
END_REGION

REGION Network 4: Verwerking iRejectSenCilUp_g0
   "ID_Reject_CM_DI_iRejectSenCilUp_g0"(iSen := "iRejectSenCilUp_g0",   // "FB_CM_DI_Sensor"
                           oSen_TON_TOF => "DB_IO".reject.iRejectSenCilUp);
END_REGION

REGION Network 5: Verwerking iRejectSenVacuum_V+
   "ID_Reject_CM_DI_iRejectSenVacuum_V+"(iSen := "iRejectSenVacuum_V+",   // "FB_CM_DI_Sensor"
                           oSen_TON_TOF => "DB_IO".reject.iRejectSenVacuum);
END_REGION

REGION Network 6: ------------------------------------------------------------------------ Logic ------------------------------------------------------------------------
END_REGION

REGION Network 7: Grafcet Reject
   IF "DB_Testing".enable.Reject THEN
       "ID_PE_Reject"(i_Init := "DB_Global".reject.init OR "DB_Testing".init.Reject,   // "FB_PE_Reject"
                      i_Enable := NOT "DB_Global".general.man AND NOT "DB_Alarm".general.global,
                      i_CmdReject := "DB_Global".reject.cmdReject OR "DB_Testing".cmd.Reject,
                      i_CoverRejectBit := "DB_Global".plate.currentCovers[6].reject OR "DB_Testing".value.RejectBit,
                      iSenCilIn := "DB_IO".reject.iRejectSenCilIn,
                      iSenCilOut := "DB_IO".reject.iRejectSenCilOut,
                      iSenCilUp := "DB_IO".reject.iRejectSenCilUp,
                      iSenVacuum := "DB_IO".reject.iRejectSenVacuum,
                      o_ReadyToReject => "DB_Global".reject.sigReadyToReject,
                      o_EmptyRejectedCoverProperties => "DB_Global".plate.currentCovers[6],
                      o_AlmVacuum => "DB_Alarm".reject.vacuum,
                      oVenCilOut => "DB_IO".reject.oRejectVenCilOut,
                      oVenCilIn => "DB_IO".reject.oRejectVenCilIn,
                      oVenCilDown => "DB_IO".reject.oRejectVenCilDown,
                      oVenVacuum => "DB_IO".reject.oRejectVenVacuum);
   END_IF;
END_REGION

REGION Network 8: ---------------------------------------------------------------------- Outputs ----------------------------------------------------------------------
END_REGION

REGION Network 9: Sturen oRejectVenCil
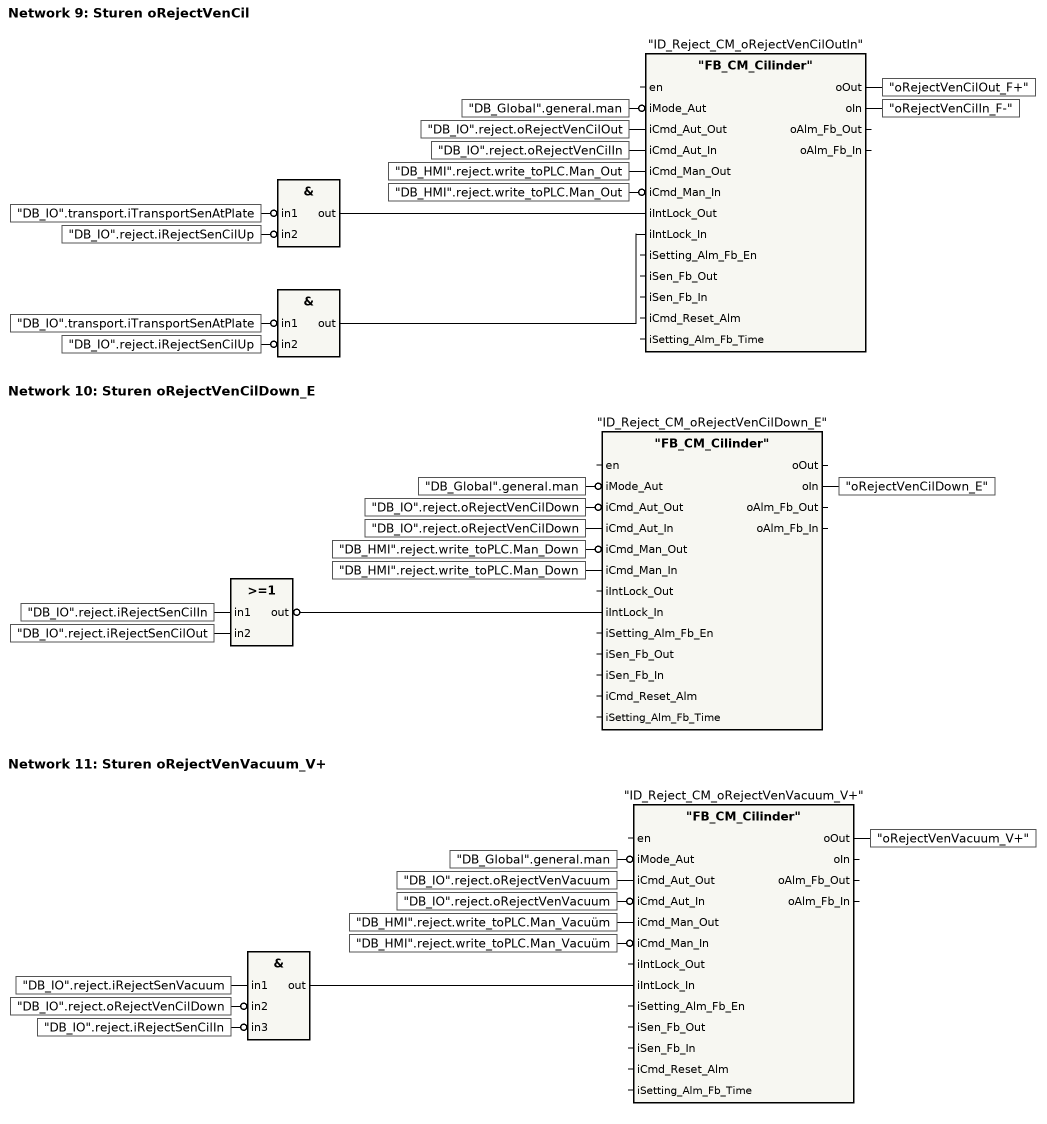
   "ID_Reject_CM_oRejectVenCilOutIn"(iMode_Aut := NOT "DB_Global".general.man,   // "FB_CM_Cilinder"
                           iCmd_Aut_Out := "DB_IO".reject.oRejectVenCilOut,
                           iCmd_Aut_In := "DB_IO".reject.oRejectVenCilIn,
                           iCmd_Man_Out := "DB_HMI".reject.write_toPLC.Man_Out,
                           iCmd_Man_In := NOT "DB_HMI".reject.write_toPLC.Man_Out,
                           iIntLock_Out := NOT "DB_IO".transport.iTransportSenAtPlate AND NOT "DB_IO".reject.iRejectSenCilUp,
                           iIntLock_In := NOT "DB_IO".transport.iTransportSenAtPlate AND NOT "DB_IO".reject.iRejectSenCilUp,
                           oOut => "oRejectVenCilOut_F+",
                           oIn => "oRejectVenCilIn_F-");
END_REGION

REGION Network 10: Sturen oRejectVenCilDown_E
   "ID_Reject_CM_oRejectVenCilDown_E"(iMode_Aut := NOT "DB_Global".general.man,   // "FB_CM_Cilinder"
                           iCmd_Aut_Out := NOT "DB_IO".reject.oRejectVenCilDown,
                           iCmd_Aut_In := "DB_IO".reject.oRejectVenCilDown,
                           iCmd_Man_Out := NOT "DB_HMI".reject.write_toPLC.Man_Down,
                           iCmd_Man_In := "DB_HMI".reject.write_toPLC.Man_Down,
                           iIntLock_In := NOT ("DB_IO".reject.iRejectSenCilIn OR "DB_IO".reject.iRejectSenCilOut),
                           oIn => "oRejectVenCilDown_E");
END_REGION

REGION Network 11: Sturen oRejectVenVacuum_V+
   // TODO:
   // - Check interlock
   "ID_Reject_CM_oRejectVenVacuum_V+"(iMode_Aut := NOT "DB_Global".general.man,   // "FB_CM_Cilinder"
                           iCmd_Aut_Out := "DB_IO".reject.oRejectVenVacuum,
                           iCmd_Aut_In := NOT "DB_IO".reject.oRejectVenVacuum,
                           iCmd_Man_Out := "DB_HMI".reject.write_toPLC.Man_Vacuüm,
                           iCmd_Man_In := NOT "DB_HMI".reject.write_toPLC.Man_Vacuüm,
                           iIntLock_In := "DB_IO".reject.iRejectSenVacuum AND NOT "DB_IO".reject.oRejectVenCilDown AND NOT "DB_IO".reject.iRejectSenCilIn,
                           oOut => "oRejectVenVacuum_V+");
END_REGION
END_FUNCTION

FUNCTION_BLOCK "FB_PE_Reject"
{ S7_Optimized_Access := 'TRUE' }
VERSION : 0.1
   VAR_INPUT 
      i_Init : Bool;
      i_Enable : Bool;
      i_CmdReject : Bool;
      i_CoverRejectBit : Bool;
      iSenCilIn : Bool;
      iSenCilOut : Bool;
      iSenCilUp : Bool;
      iSenVacuum : Bool;
   END_VAR

   VAR_OUTPUT 
      o_ReadyToReject : Bool;
      o_EmptyRejectedCoverProperties : "UDT_coverProperties";
      o_AlmVacuum : Bool;   // Indicates that the item fell during reject proces
      oVenCilOut : Bool;   // Bistable
      oVenCilIn : Bool;   // Bistable
      oVenCilDown : Bool;
      oVenVacuum : Bool;
   END_VAR

   VAR 
      sStep : Int;
      sInit : Bool;
      sPreviuousStep : Int;
      sTON_X1 {InstructionName := 'TON_TIME'; LibVersion := '1.0'} : TON_TIME;
      sTON_X2 {InstructionName := 'TON_TIME'; LibVersion := '1.0'} : TON_TIME;
      sTON_X3 {InstructionName := 'TON_TIME'; LibVersion := '1.0'} : TON_TIME;
      sTON_X4 {InstructionName := 'TON_TIME'; LibVersion := '1.0'} : TON_TIME;
      sTON_X5 {InstructionName := 'TON_TIME'; LibVersion := '1.0'} : TON_TIME;
      sTON_X6 {InstructionName := 'TON_TIME'; LibVersion := '1.0'} : TON_TIME;
      sTON_X7 {InstructionName := 'TON_TIME'; LibVersion := '1.0'} : TON_TIME;
      sTON_X8 {InstructionName := 'TON_TIME'; LibVersion := '1.0'} : TON_TIME;
      sTON_X9 {InstructionName := 'TON_TIME'; LibVersion := '1.0'} : TON_TIME;
   END_VAR

   VAR CONSTANT 
      cShortWaitTime : Time := T#0.5s;   // With feedback
      cLongWaitTime : Time := T#1.5s;   // Without feedback
      cPulseWaitTime : Time := T#100ms;   // Pulse for bistable valve
   END_VAR


BEGIN
	REGION init
	    IF #i_Init AND NOT (#sInit = #i_Init) THEN
	        #sStep := 0;
	    END_IF;
	    #sInit := #i_Init;
	END_REGION
	
	REGION enable
	    IF NOT #i_Enable THEN
	        GOTO afterGrafcetLogic;
	    END_IF;
	END_REGION
	
	REGION timers
	    
	    #sTON_X1(IN := #sStep = 1,
	             PT := #cPulseWaitTime);
	    
	    #sTON_X2(IN := (#sStep = 2) AND #iSenCilOut ,
	             PT := #cShortWaitTime);
	    
	    #sTON_X3(IN := (#sStep = 3) AND NOT #iSenCilOut,
	             PT := #cLongWaitTime);
	    
	    #sTON_X4(IN := (#sStep = 4) AND #iSenVacuum,
	             PT := #cShortWaitTime);
	    
	    #sTON_X5(IN := (#sStep = 5) AND #iSenCilUp,
	             PT := #cShortWaitTime);
	    
	    #sTON_X6(IN := (#sStep = 6),
	             PT := #cPulseWaitTime);
	    
	    #sTON_X7(IN := (#sStep = 7) AND #iSenCilIn,
	             PT := #cShortWaitTime);
	    
	    #sTON_X8(IN := (#sStep = 8) AND NOT #iSenCilUp,
	             PT := #cLongWaitTime);
	    
	    #sTON_X9(IN:= #sStep = 9,
	             PT:= #cShortWaitTime);
	    
	END_REGION
	
	REGION grafcet logic
	    CASE #sStep OF
	        0:
	            IF
	                #i_CmdReject
	                AND #i_CoverRejectBit
	                AND #iSenCilIn
	                AND #iSenCilUp
	            THEN
	                #sStep := 1;
	            END_IF;
	        1:
	            IF #sTON_X1.Q THEN
	                #sStep := 2;
	            END_IF;
	        2:
	            IF #sTON_X2.Q THEN
	                #sStep := 3;
	            END_IF;
	        3:
	            IF #sTON_X3.Q THEN
	                #sStep := 4;
	            END_IF;
	        4:
	            IF #sTON_X4.Q THEN
	                #sStep := 5;
	            END_IF;
	        5:
	            IF #sTON_X5.Q THEN
	                #sStep := 6;
	            END_IF;
	        6:
	            IF #sTON_X6.Q THEN
	                #sStep := 7;
	            END_IF;
	        7:
	            IF #sTON_X7.Q THEN
	                #sStep := 8;
	            END_IF;
	        8:
	            IF #sTON_X8.Q THEN
	                #sStep := 9;
	            END_IF;
	        9:
	            IF #sTON_X9.Q THEN
	                #sStep := 0;
	            END_IF;
	        ELSE
	            #sStep := 0;
	    END_CASE;
	END_REGION
	
	afterGrafcetLogic: // Jump destination
	
	REGION empty rejected cover properties
	    
	    IF
	        (#sStep = 7)
	        AND NOT (#sPreviuousStep = #sStep)
	    THEN
	        #o_EmptyRejectedCoverProperties := "FC_emptyCoverProperties"();
	    END_IF;
	    
	    #sPreviuousStep := #sStep;
	    
	END_REGION
	
	REGION alarm item fell during reject
	    
	    IF #sStep >= 5 AND #sStep <= 8 AND NOT #iSenVacuum THEN
	        #o_AlmVacuum := TRUE;
	    ELSE
	        #o_AlmVacuum := FALSE;
	    END_IF;
	    
	END_REGION
	
	REGION outputs
	    
	    #o_ReadyToReject := #sStep = 0;
	    
	    #oVenCilOut      := #sStep = 1;
	    
	    #oVenCilIn       := #sStep = 6;
	    
	    #oVenCilDown     := #sStep = 3
	                     OR #sStep = 4
	                     OR #sStep = 8
	                     OR #sStep = 9;
	                     
	    #oVenVacuum      := #sStep = 4
	                     OR #sStep = 5
	                     OR #sStep = 6
	                     OR #sStep = 7
	                     OR #sStep = 8;
	                     
	END_REGION
	
END_FUNCTION_BLOCK

FUNCTION "FC_emptyCoverProperties" : "UDT_coverProperties"
{ S7_Optimized_Access := 'TRUE' }
VERSION : 0.1
   VAR_TEMP 
      xEmptyCover : "UDT_coverProperties";
   END_VAR


BEGIN
	#xEmptyCover.loaded := FALSE;
	#xEmptyCover.reject := FALSE;
	#xEmptyCover.properties.correctOrientation := FALSE;
	#xEmptyCover.properties.metallic := FALSE;
	#xEmptyCover.properties.notBlack := FALSE;
	
	#FC_emptyCoverProperties := #xEmptyCover;
END_FUNCTION

FUNCTION "FC_EM_Transport" : Void   // FC6, FBD
{ S7_Optimized_Access := 'TRUE' }
// stored: SetENOAutomatically false
BEGIN

REGION Network 1: ------------------------------------------------------------------------ Inputs ------------------------------------------------------------------------
END_REGION

REGION Network 2: Verwerking iTransportSenDown_h1
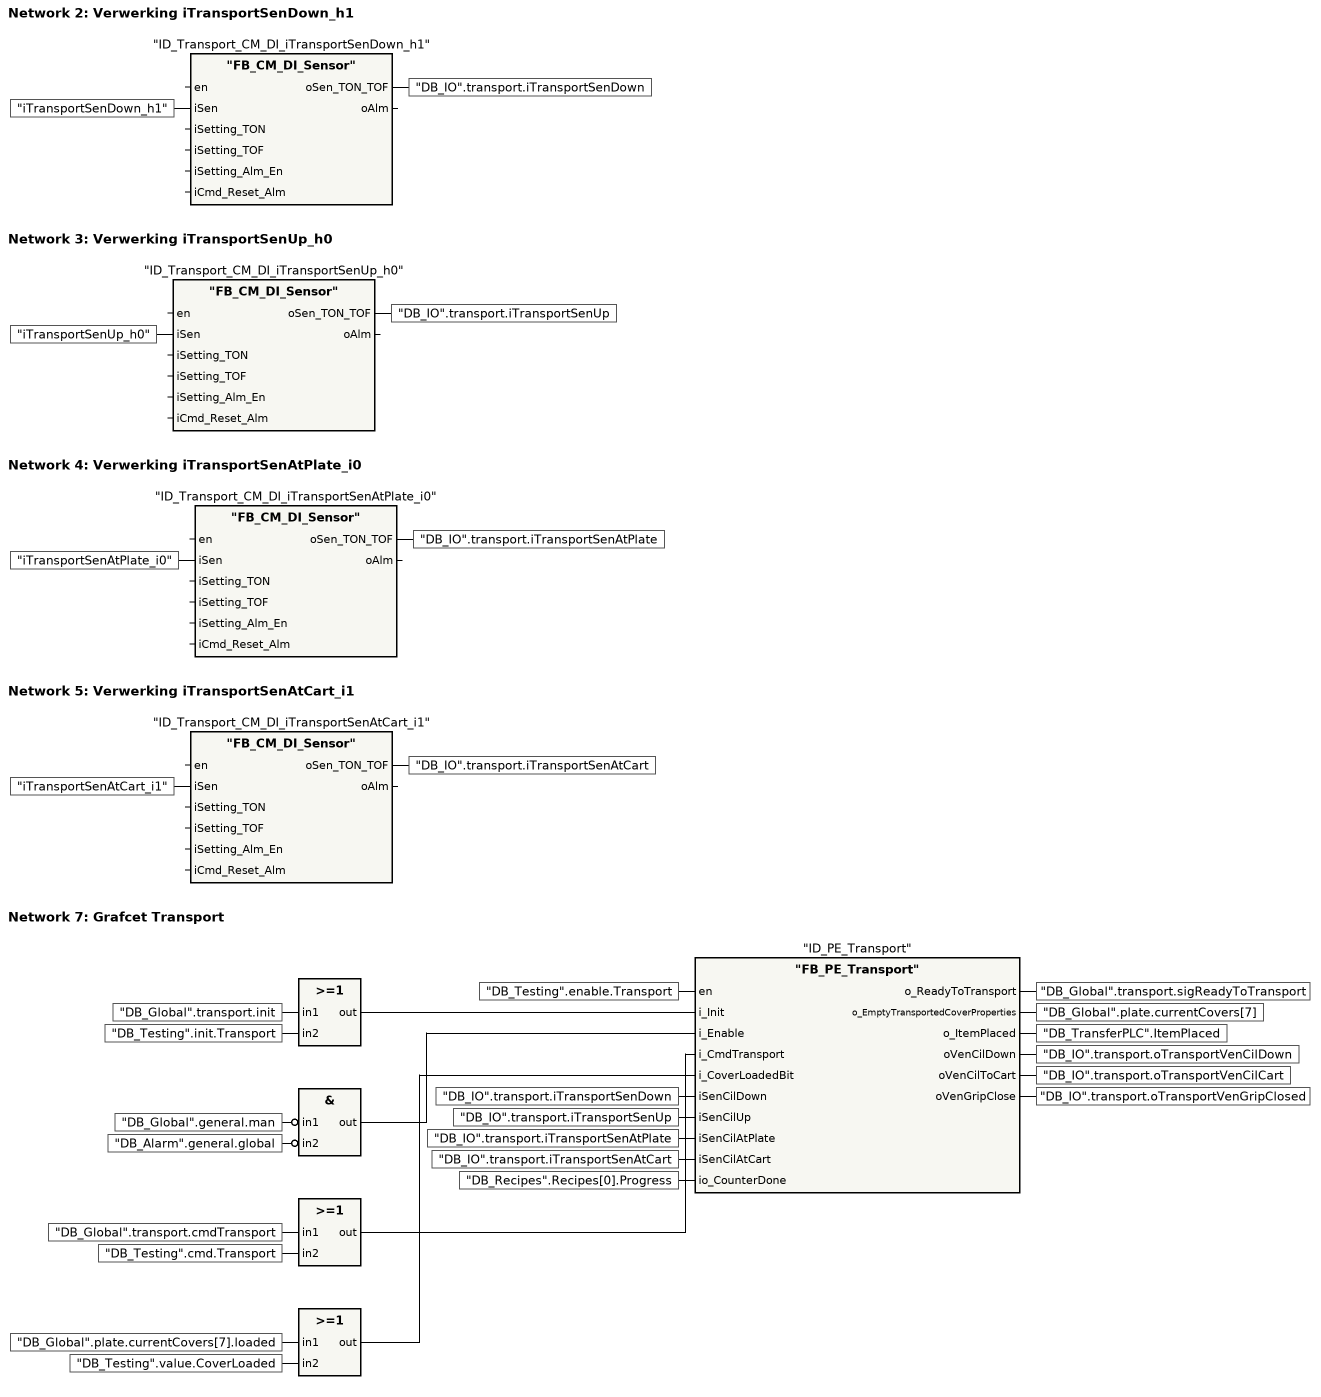
   "ID_Transport_CM_DI_iTransportSenDown_h1"(iSen := "iTransportSenDown_h1",   // "FB_CM_DI_Sensor"
                           oSen_TON_TOF => "DB_IO".transport.iTransportSenDown);
END_REGION

REGION Network 3: Verwerking iTransportSenUp_h0
   "ID_Transport_CM_DI_iTransportSenUp_h0"(iSen := "iTransportSenUp_h0",   // "FB_CM_DI_Sensor"
                           oSen_TON_TOF => "DB_IO".transport.iTransportSenUp);
END_REGION

REGION Network 4: Verwerking iTransportSenAtPlate_i0
   "ID_Transport_CM_DI_iTransportSenAtPlate_i0"(iSen := "iTransportSenAtPlate_i0",   // "FB_CM_DI_Sensor"
                           oSen_TON_TOF => "DB_IO".transport.iTransportSenAtPlate);
END_REGION

REGION Network 5: Verwerking iTransportSenAtCart_i1
   "ID_Transport_CM_DI_iTransportSenAtCart_i1"(iSen := "iTransportSenAtCart_i1",   // "FB_CM_DI_Sensor"
                           oSen_TON_TOF => "DB_IO".transport.iTransportSenAtCart);
END_REGION

REGION Network 6: ------------------------------------------------------------------------ Logic ------------------------------------------------------------------------
END_REGION

